LIN {X 29.26, Y 198.76, Z 40.25, A 0, B 90, C 0, E1 0, E2 0, E3 0, E4 0} C_DIS
LIN {X 27.26, Y 190.891, Z 40.25, A 0, B 90, C 0, E1 0, E2 0, E3 0, E4 0} C_DIS
LIN {X 25.335, Y 183.004, Z 40.25, A 0, B 90, C 0, E1 0, E2 0, E3 0, E4 0} C_DIS
LIN {X 23.484, Y 175.099, Z 40.25, A 0, B 90, C 0, E1 0, E2 0, E3 0, E4 0} C_DIS
LIN {X 21.71, Y 167.176, Z 40.25, A 0, B 90, C 0, E1 0, E2 0, E3 0, E4 0} C_DIS
LIN {X 20.012, Y 159.237, Z 40.25, A 0, B 90, C 0, E1 0, E2 0, E3 0, E4 0} C_DIS
LIN {X 18.392, Y 151.282, Z 40.25, A 0, B 90, C 0, E1 0, E2 0, E3 0, E4 0} C_DIS
LIN {X 16.851, Y 143.31, Z 40.25, A 0, B 90, C 0, E1 0, E2 0, E3 0, E4 0} C_DIS
LIN {X 15.39, Y 135.324, Z 40.25, A 0, B 90, C 0, E1 0, E2 0, E3 0, E4 0} C_DIS
LIN {X 14.009, Y 127.324, Z 40.25, A 0, B 90, C 0, E1 0, E2 0, E3 0, E4 0} C_DIS
LIN {X 12.709, Y 119.309, Z 40.25, A 0, B 90, C 0, E1 0, E2 0, E3 0, E4 0} C_DIS
LIN {X 11.491, Y 111.283, Z 40.25, A 0, B 90, C 0, E1 0, E2 0, E3 0, E4 0} C_DIS
LIN {X 10.355, Y 103.244, Z 40.25, A 0, B 90, C 0, E1 0, E2 0, E3 0, E4 0} C_DIS
LIN {X 9.301, Y 95.193, Z 40.25, A 0, B 90, C 0, E1 0, E2 0, E3 0, E4 0} C_DIS
LIN {X 8.331, Y 87.133, Z 40.25, A 0, B 90, C 0, E1 0, E2 0, E3 0, E4 0} C_DIS
LIN {X 7.444, Y 79.063, Z 40.25, A 0, B 90, C 0, E1 0, E2 0, E3 0, E4 0} C_DIS
LIN {X 6.642, Y 70.983, Z 40.25, A 0, B 90, C 0, E1 0, E2 0, E3 0, E4 0} C_DIS
LIN {X 5.924, Y 62.896, Z 40.25, A 0, B 90, C 0, E1 0, E2 0, E3 0, E4 0} C_DIS
LIN {X 5.292, Y 54.802, Z 40.25, A 0, B 90, C 0, E1 0, E2 0, E3 0, E4 0} C_DIS
LIN {X 4.746, Y 46.702, Z 40.25, A 0, B 90, C 0, E1 0, E2 0, E3 0, E4 0} C_DIS
LIN {X 4.285, Y 38.596, Z 40.25, A 0, B 90, C 0, E1 0, E2 0, E3 0, E4 0} C_DIS
LIN {X 3.911, Y 30.486, Z 40.25, A 0, B 90, C 0, E1 0, E2 0, E3 0, E4 0} C_DIS
LIN {X 3.624, Y 22.372, Z 40.25, A 0, B 90, C 0, E1 0, E2 0, E3 0, E4 0} C_DIS
LIN {X 3.424, Y 14.256, Z 40.25, A 0, B 90, C 0, E1 0, E2 0, E3 0, E4 0} C_DIS
LIN {X 3.313, Y 6.138, Z 40.25, A 0, B 90, C 0, E1 0, E2 0, E3 0, E4 0} C_DIS
LIN {X 3.289, Y -1.981, Z 40.25, A 0, B 90, C 0, E1 0, E2 0, E3 0, E4 0} C_DIS
LIN {X 3.353, Y -10.1, Z 40.25, A 0, B 90, C 0, E1 0, E2 0, E3 0, E4 0} C_DIS
LIN {X 3.506, Y -18.217, Z 40.25, A 0, B 90, C 0, E1 0, E2 0, E3 0, E4 0} C_DIS
LIN {X 3.747, Y -26.332, Z 40.25, A 0, B 90, C 0, E1 0, E2 0, E3 0, E4 0} C_DIS
LIN {X 4.074, Y -34.444, Z 40.25, A 0, B 90, C 0, E1 0, E2 0, E3 0, E4 0} C_DIS
LIN {X 4.489, Y -42.553, Z 40.25, A 0, B 90, C 0, E1 0, E2 0, E3 0, E4 0} C_DIS
LIN {X 4.99, Y -50.656, Z 40.25, A 0, B 90, C 0, E1 0, E2 0, E3 0, E4 0} C_DIS
LIN {X 5.578, Y -58.754, Z 40.25, A 0, B 90, C 0, E1 0, E2 0, E3 0, E4 0} C_DIS
LIN {X 6.252, Y -66.844, Z 40.25, A 0, B 90, C 0, E1 0, E2 0, E3 0, E4 0} C_DIS
LIN {X 7.011, Y -74.928, Z 40.25, A 0, B 90, C 0, E1 0, E2 0, E3 0, E4 0} C_DIS
LIN {X 7.855, Y -83.002, Z 40.25, A 0, B 90, C 0, E1 0, E2 0, E3 0, E4 0} C_DIS
LIN {X 8.784, Y -91.068, Z 40.25, A 0, B 90, C 0, E1 0, E2 0, E3 0, E4 0} C_DIS
LIN {X 9.797, Y -99.123, Z 40.25, A 0, B 90, C 0, E1 0, E2 0, E3 0, E4 0} C_DIS
LIN {X 10.893, Y -107.168, Z 40.25, A 0, B 90, C 0, E1 0, E2 0, E3 0, E4 0} C_DIS
LIN {X 12.071, Y -115.201, Z 40.25, A 0, B 90, C 0, E1 0, E2 0, E3 0, E4 0} C_DIS
LIN {X 13.332, Y -123.221, Z 40.25, A 0, B 90, C 0, E1 0, E2 0, E3 0, E4 0} C_DIS
LIN {X 14.674, Y -131.228, Z 40.25, A 0, B 90, C 0, E1 0, E2 0, E3 0, E4 0} C_DIS
LIN {X 16.096, Y -139.221, Z 40.25, A 0, B 90, C 0, E1 0, E2 0, E3 0, E4 0} C_DIS
LIN {X 17.599, Y -147.2, Z 40.25, A 0, B 90, C 0, E1 0, E2 0, E3 0, E4 0} C_DIS
LIN {X 19.18, Y -155.163, Z 40.25, A 0, B 90, C 0, E1 0, E2 0, E3 0, E4 0} C_DIS
LIN {X 20.84, Y -163.111, Z 40.25, A 0, B 90, C 0, E1 0, E2 0, E3 0, E4 0} C_DIS
LIN {X 22.577, Y -171.042, Z 40.25, A 0, B 90, C 0, E1 0, E2 0, E3 0, E4 0} C_DIS
LIN {X 24.389, Y -178.956, Z 40.25, A 0, B 90, C 0, E1 0, E2 0, E3 0, E4 0} C_DIS
LIN {X 26.277, Y -186.852, Z 40.25, A 0, B 90, C 0, E1 0, E2 0, E3 0, E4 0} C_DIS
LIN {X 28.238, Y -194.73, Z 40.25, A 0, B 90, C 0, E1 0, E2 0, E3 0, E4 0} C_DIS
LIN {X 30.272, Y -202.59, Z 40.25, A 0, B 90, C 0, E1 0, E2 0, E3 0, E4 0} C_DIS
LIN {X 32.378, Y -210.431, Z 40.25, A 0, B 90, C 0, E1 0, E2 0, E3 0, E4 0} C_DIS
LIN {X 34.554, Y -218.253, Z 40.25, A 0, B 90, C 0, E1 0, E2 0, E3 0, E4 0} C_DIS
LIN {X 36.8, Y -226.055, Z 40.25, A 0, B 90, C 0, E1 0, E2 0, E3 0, E4 0} C_DIS
LIN {X 39.114, Y -233.837, Z 40.25, A 0, B 90, C 0, E1 0, E2 0, E3 0, E4 0} C_DIS
LIN {X 41.496, Y -241.599, Z 40.25, A 0, B 90, C 0, E1 0, E2 0, E3 0, E4 0} C_DIS
LIN {X 43.943, Y -249.34, Z 40.25, A 0, B 90, C 0, E1 0, E2 0, E3 0, E4 0} C_DIS
LIN {X 46.455, Y -257.06, Z 40.25, A 0, B 90, C 0, E1 0, E2 0, E3 0, E4 0} C_DIS
LIN {X 49.031, Y -264.76, Z 40.25, A 0, B 90, C 0, E1 0, E2 0, E3 0, E4 0} C_DIS
LIN {X 51.67, Y -272.438, Z 40.25, A 0, B 90, C 0, E1 0, E2 0, E3 0, E4 0} C_DIS
LIN {X 54.369, Y -280.094, Z 40.25, A 0, B 90, C 0, E1 0, E2 0, E3 0, E4 0} C_DIS
LIN {X 57.13, Y -287.73, Z 40.25, A 0, B 90, C 0, E1 0, E2 0, E3 0, E4 0} C_DIS
LIN {X 59.951, Y -295.342, Z 40.25, A 0, B 90, C 0, E1 0, E2 0, E3 0, E4 0} C_DIS
LIN {X 62.833, Y -302.932, Z 40.25, A 0, B 90, C 0, E1 0, E2 0, E3 0, E4 0} C_DIS
LIN {X 65.777, Y -310.499, Z 40.25, A 0, B 90, C 0, E1 0, E2 0, E3 0, E4 0} C_DIS
LIN {X 68.781, Y -318.042, Z 40.25, A 0, B 90, C 0, E1 0, E2 0, E3 0, E4 0} C_DIS
LIN {X 71.847, Y -325.559, Z 40.25, A 0, B 90, C 0, E1 0, E2 0, E3 0, E4 0} C_DIS
LIN {X 74.973, Y -333.052, Z 40.25, A 0, B 90, C 0, E1 0, E2 0, E3 0, E4 0} C_DIS
LIN {X 78.074, Y -340.551, Z 40.25, A 0, B 90, C 0, E1 0, E2 0, E3 0, E4 0} C_DIS
LIN {X 75.376, Y -347.755, Z 40.25, A 0, B 90, C 0, E1 0, E2 0, E3 0, E4 0} C_DIS
LIN {X 68.14, Y -351.37, Z 40.25, A 0, B 90, C 0, E1 0, E2 0, E3 0, E4 0} C_DIS
LIN {X 60.675, Y -354.562, Z 40.25, A 0, B 90, C 0, E1 0, E2 0, E3 0, E4 0} C_DIS
LIN {X 53.21, Y -357.754, Z 40.25, A 0, B 90, C 0, E1 0, E2 0, E3 0, E4 0} C_DIS
LIN {X 45.745, Y -360.947, Z 40.25, A 0, B 90, C 0, E1 0, E2 0, E3 0, E4 0} C_DIS
LIN {X 38.28, Y -364.139, Z 40.25, A 0, B 90, C 0, E1 0, E2 0, E3 0, E4 0} C_DIS
LIN {X 30.815, Y -367.331, Z 40.25, A 0, B 90, C 0, E1 0, E2 0, E3 0, E4 0} C_DIS
LIN {X 23.35, Y -370.523, Z 40.25, A 0, B 90, C 0, E1 0, E2 0, E3 0, E4 0} C_DIS
LIN {X 15.615, Y -372.622, Z 40.25, A 0, B 90, C 0, E1 0, E2 0, E3 0, E4 0} C_DIS
LIN {X 9.092, Y -368.331, Z 40.25, A 0, B 90, C 0, E1 0, E2 0, E3 0, E4 0} C_DIS
LIN {X 5.884, Y -360.875, Z 40.25, A 0, B 90, C 0, E1 0, E2 0, E3 0, E4 0} C_DIS
LIN {X 2.773, Y -353.376, Z 40.25, A 0, B 90, C 0, E1 0, E2 0, E3 0, E4 0} C_DIS
LIN {X -0.284, Y -345.854, Z 40.25, A 0, B 90, C 0, E1 0, E2 0, E3 0, E4 0} C_DIS
LIN {X -3.286, Y -338.311, Z 40.25, A 0, B 90, C 0, E1 0, E2 0, E3 0, E4 0} C_DIS
LIN {X -6.234, Y -330.746, Z 40.25, A 0, B 90, C 0, E1 0, E2 0, E3 0, E4 0} C_DIS
LIN {X -9.127, Y -323.16, Z 40.25, A 0, B 90, C 0, E1 0, E2 0, E3 0, E4 0} C_DIS
LIN {X -11.965, Y -315.554, Z 40.25, A 0, B 90, C 0, E1 0, E2 0, E3 0, E4 0} C_DIS
LIN {X -14.749, Y -307.927, Z 40.25, A 0, B 90, C 0, E1 0, E2 0, E3 0, E4 0} C_DIS
LIN {X -17.478, Y -300.281, Z 40.25, A 0, B 90, C 0, E1 0, E2 0, E3 0, E4 0} C_DIS
LIN {X -20.15, Y -292.614, Z 40.25, A 0, B 90, C 0, E1 0, E2 0, E3 0, E4 0} C_DIS
LIN {X -22.764, Y -284.928, Z 40.25, A 0, B 90, C 0, E1 0, E2 0, E3 0, E4 0} C_DIS
LIN {X -25.32, Y -277.221, Z 40.25, A 0, B 90, C 0, E1 0, E2 0, E3 0, E4 0} C_DIS
LIN {X -27.815, Y -269.496, Z 40.25, A 0, B 90, C 0, E1 0, E2 0, E3 0, E4 0} C_DIS
LIN {X -30.249, Y -261.75, Z 40.25, A 0, B 90, C 0, E1 0, E2 0, E3 0, E4 0} C_DIS
LIN {X -32.621, Y -253.986, Z 40.25, A 0, B 90, C 0, E1 0, E2 0, E3 0, E4 0} C_DIS
LIN {X -34.93, Y -246.202, Z 40.25, A 0, B 90, C 0, E1 0, E2 0, E3 0, E4 0} C_DIS
LIN {X -37.174, Y -238.399, Z 40.25, A 0, B 90, C 0, E1 0, E2 0, E3 0, E4 0} C_DIS
LIN {X -39.353, Y -230.578, Z 40.25, A 0, B 90, C 0, E1 0, E2 0, E3 0, E4 0} C_DIS
LIN {X -41.465, Y -222.739, Z 40.25, A 0, B 90, C 0, E1 0, E2 0, E3 0, E4 0} C_DIS
LIN {X -43.512, Y -214.883, Z 40.25, A 0, B 90, C 0, E1 0, E2 0, E3 0, E4 0} C_DIS
LIN {X -45.49, Y -207.009, Z 40.25, A 0, B 90, C 0, E1 0, E2 0, E3 0, E4 0} C_DIS
LIN {X -47.401, Y -199.118, Z 40.25, A 0, B 90, C 0, E1 0, E2 0, E3 0, E4 0} C_DIS
LIN {X -49.243, Y -191.211, Z 40.25, A 0, B 90, C 0, E1 0, E2 0, E3 0, E4 0} C_DIS
LIN {X -51.015, Y -183.288, Z 40.25, A 0, B 90, C 0, E1 0, E2 0, E3 0, E4 0} C_DIS
LIN {X -52.717, Y -175.349, Z 40.25, A 0, B 90, C 0, E1 0, E2 0, E3 0, E4 0} C_DIS
LIN {X -54.348, Y -167.396, Z 40.25, A 0, B 90, C 0, E1 0, E2 0, E3 0, E4 0} C_DIS
LIN {X -55.907, Y -159.428, Z 40.25, A 0, B 90, C 0, E1 0, E2 0, E3 0, E4 0} C_DIS
LIN {X -57.394, Y -151.446, Z 40.25, A 0, B 90, C 0, E1 0, E2 0, E3 0, E4 0} C_DIS
LIN {X -58.807, Y -143.452, Z 40.25, A 0, B 90, C 0, E1 0, E2 0, E3 0, E4 0} C_DIS
LIN {X -60.147, Y -135.444, Z 40.25, A 0, B 90, C 0, E1 0, E2 0, E3 0, E4 0} C_DIS
LIN {X -61.412, Y -127.424, Z 40.25, A 0, B 90, C 0, E1 0, E2 0, E3 0, E4 0} C_DIS
LIN {X -62.602, Y -119.393, Z 40.25, A 0, B 90, C 0, E1 0, E2 0, E3 0, E4 0} C_DIS
LIN {X -63.717, Y -111.351, Z 40.25, A 0, B 90, C 0, E1 0, E2 0, E3 0, E4 0} C_DIS
LIN {X -64.755, Y -103.299, Z 40.25, A 0, B 90, C 0, E1 0, E2 0, E3 0, E4 0} C_DIS
LIN {X -65.718, Y -95.238, Z 40.25, A 0, B 90, C 0, E1 0, E2 0, E3 0, E4 0} C_DIS
LIN {X -66.604, Y -87.167, Z 40.25, A 0, B 90, C 0, E1 0, E2 0, E3 0, E4 0} C_DIS
LIN {X -67.412, Y -79.089, Z 40.25, A 0, B 90, C 0, E1 0, E2 0, E3 0, E4 0} C_DIS
LIN {X -68.144, Y -71.003, Z 40.25, A 0, B 90, C 0, E1 0, E2 0, E3 0, E4 0} C_DIS
LIN {X -68.798, Y -62.911, Z 40.25, A 0, B 90, C 0, E1 0, E2 0, E3 0, E4 0} C_DIS
LIN {X -69.374, Y -54.812, Z 40.25, A 0, B 90, C 0, E1 0, E2 0, E3 0, E4 0} C_DIS
LIN {X -69.872, Y -46.709, Z 40.25, A 0, B 90, C 0, E1 0, E2 0, E3 0, E4 0} C_DIS
LIN {X -70.291, Y -38.601, Z 40.25, A 0, B 90, C 0, E1 0, E2 0, E3 0, E4 0} C_DIS
LIN {X -70.631, Y -30.489, Z 40.25, A 0, B 90, C 0, E1 0, E2 0, E3 0, E4 0} C_DIS
LIN {X -70.892, Y -22.374, Z 40.25, A 0, B 90, C 0, E1 0, E2 0, E3 0, E4 0} C_DIS
LIN {X -71.073, Y -14.257, Z 40.25, A 0, B 90, C 0, E1 0, E2 0, E3 0, E4 0} C_DIS
LIN {X -71.174, Y -6.139, Z 40.25, A 0, B 90, C 0, E1 0, E2 0, E3 0, E4 0} C_DIS
LIN {X -71.195, Y 1.979, Z 40.25, A 0, B 90, C 0, E1 0, E2 0, E3 0, E4 0} C_DIS
LIN {X -71.136, Y 10.098, Z 40.25, A 0, B 90, C 0, E1 0, E2 0, E3 0, E4 0} C_DIS
LIN {X -70.996, Y 18.216, Z 40.25, A 0, B 90, C 0, E1 0, E2 0, E3 0, E4 0} C_DIS
LIN {X -70.777, Y 26.332, Z 40.25, A 0, B 90, C 0, E1 0, E2 0, E3 0, E4 0} C_DIS
LIN {X -70.478, Y 34.445, Z 40.25, A 0, B 90, C 0, E1 0, E2 0, E3 0, E4 0} C_DIS
LIN {X -70.099, Y 42.555, Z 40.25, A 0, B 90, C 0, E1 0, E2 0, E3 0, E4 0} C_DIS
LIN {X -69.642, Y 50.661, Z 40.25, A 0, B 90, C 0, E1 0, E2 0, E3 0, E4 0} C_DIS
LIN {X -69.107, Y 58.762, Z 40.25, A 0, B 90, C 0, E1 0, E2 0, E3 0, E4 0} C_DIS
LIN {X -68.493, Y 66.858, Z 40.25, A 0, B 90, C 0, E1 0, E2 0, E3 0, E4 0} C_DIS
LIN {X -67.801, Y 74.947, Z 40.25, A 0, B 90, C 0, E1 0, E2 0, E3 0, E4 0} C_DIS
LIN {X -67.031, Y 83.029, Z 40.25, A 0, B 90, C 0, E1 0, E2 0, E3 0, E4 0} C_DIS
LIN {X -66.184, Y 91.104, Z 40.25, A 0, B 90, C 0, E1 0, E2 0, E3 0, E4 0} C_DIS
LIN {X -65.26, Y 99.17, Z 40.25, A 0, B 90, C 0, E1 0, E2 0, E3 0, E4 0} C_DIS
LIN {X -64.26, Y 107.227, Z 40.25, A 0, B 90, C 0, E1 0, E2 0, E3 0, E4 0} C_DIS
LIN {X -63.183, Y 115.274, Z 40.25, A 0, B 90, C 0, E1 0, E2 0, E3 0, E4 0} C_DIS
LIN {X -62.031, Y 123.311, Z 40.25, A 0, B 90, C 0, E1 0, E2 0, E3 0, E4 0} C_DIS
LIN {X -60.803, Y 131.336, Z 40.25, A 0, B 90, C 0, E1 0, E2 0, E3 0, E4 0} C_DIS
LIN {X -59.501, Y 139.35, Z 40.25, A 0, B 90, C 0, E1 0, E2 0, E3 0, E4 0} C_DIS
LIN {X -58.125, Y 147.351, Z 40.25, A 0, B 90, C 0, E1 0, E2 0, E3 0, E4 0} C_DIS
LIN {X -56.675, Y 155.339, Z 40.25, A 0, B 90, C 0, E1 0, E2 0, E3 0, E4 0} C_DIS
LIN {X -55.153, Y 163.314, Z 40.25, A 0, B 90, C 0, E1 0, E2 0, E3 0, E4 0} C_DIS
LIN {X -53.558, Y 171.275, Z 40.25, A 0, B 90, C 0, E1 0, E2 0, E3 0, E4 0} C_DIS
LIN {X -51.893, Y 179.221, Z 40.25, A 0, B 90, C 0, E1 0, E2 0, E3 0, E4 0} C_DIS
LIN {X -50.157, Y 187.152, Z 40.25, A 0, B 90, C 0, E1 0, E2 0, E3 0, E4 0} C_DIS
LIN {X -48.351, Y 195.068, Z 40.25, A 0, B 90, C 0, E1 0, E2 0, E3 0, E4 0} C_DIS
LIN {X -46.476, Y 202.967, Z 40.25, A 0, B 90, C 0, E1 0, E2 0, E3 0, E4 0} C_DIS
LIN {X -44.533, Y 210.85, Z 40.25, A 0, B 90, C 0, E1 0, E2 0, E3 0, E4 0} C_DIS
LIN {X -42.521, Y 218.716, Z 40.25, A 0, B 90, C 0, E1 0, E2 0, E3 0, E4 0} C_DIS
LIN {X -40.443, Y 226.564, Z 40.25, A 0, B 90, C 0, E1 0, E2 0, E3 0, E4 0} C_DIS
LIN {X -38.298, Y 234.394, Z 40.25, A 0, B 90, C 0, E1 0, E2 0, E3 0, E4 0} C_DIS
LIN {X -36.088, Y 242.206, Z 40.25, A 0, B 90, C 0, E1 0, E2 0, E3 0, E4 0} C_DIS
LIN {X -34.098, Y 250, Z 42.75, A 0, B 90, C 0, E1 0, E2 0, E3 0, E4 0} C_DIS
LIN {X -31.758, Y 257.753, Z 42.75, A 0, B 90, C 0, E1 0, E2 0, E3 0, E4 0} C_DIS
LIN {X -29.355, Y 265.488, Z 42.75, A 0, B 90, C 0, E1 0, E2 0, E3 0, E4 0} C_DIS
LIN {X -26.891, Y 273.202, Z 42.75, A 0, B 90, C 0, E1 0, E2 0, E3 0, E4 0} C_DIS
LIN {X -24.365, Y 280.897, Z 42.75, A 0, B 90, C 0, E1 0, E2 0, E3 0, E4 0} C_DIS
LIN {X -21.781, Y 288.573, Z 42.75, A 0, B 90, C 0, E1 0, E2 0, E3 0, E4 0} C_DIS
LIN {X -19.138, Y 296.228, Z 42.75, A 0, B 90, C 0, E1 0, E2 0, E3 0, E4 0} C_DIS
LIN {X -16.439, Y 303.864, Z 42.75, A 0, B 90, C 0, E1 0, E2 0, E3 0, E4 0} C_DIS
LIN {X -13.684, Y 311.48, Z 42.75, A 0, B 90, C 0, E1 0, E2 0, E3 0, E4 0} C_DIS
LIN {X -10.874, Y 319.076, Z 42.75, A 0, B 90, C 0, E1 0, E2 0, E3 0, E4 0} C_DIS
LIN {X -8.01, Y 326.652, Z 42.75, A 0, B 90, C 0, E1 0, E2 0, E3 0, E4 0} C_DIS
LIN {X -5.092, Y 334.206, Z 42.75, A 0, B 90, C 0, E1 0, E2 0, E3 0, E4 0} C_DIS
LIN {X -2.12, Y 341.74, Z 42.75, A 0, B 90, C 0, E1 0, E2 0, E3 0, E4 0} C_DIS
LIN {X 0.906, Y 349.252, Z 42.75, A 0, B 90, C 0, E1 0, E2 0, E3 0, E4 0} C_DIS
LIN {X 3.988, Y 356.742, Z 42.75, A 0, B 90, C 0, E1 0, E2 0, E3 0, E4 0} C_DIS
LIN {X 7.123, Y 364.209, Z 42.75, A 0, B 90, C 0, E1 0, E2 0, E3 0, E4 0} C_DIS
LIN {X 11.532, Y 370.814, Z 42.75, A 0, B 90, C 0, E1 0, E2 0, E3 0, E4 0} C_DIS
LIN {X 19.315, Y 371.572, Z 42.75, A 0, B 90, C 0, E1 0, E2 0, E3 0, E4 0} C_DIS
LIN {X 26.761, Y 368.386, Z 42.75, A 0, B 90, C 0, E1 0, E2 0, E3 0, E4 0} C_DIS
LIN {X 34.207, Y 365.2, Z 42.75, A 0, B 90, C 0, E1 0, E2 0, E3 0, E4 0} C_DIS
LIN {X 41.653, Y 362.015, Z 42.75, A 0, B 90, C 0, E1 0, E2 0, E3 0, E4 0} C_DIS
LIN {X 49.099, Y 358.829, Z 42.75, A 0, B 90, C 0, E1 0, E2 0, E3 0, E4 0} C_DIS
LIN {X 56.545, Y 355.643, Z 42.75, A 0, B 90, C 0, E1 0, E2 0, E3 0, E4 0} C_DIS
LIN {X 63.991, Y 352.457, Z 42.75, A 0, B 90, C 0, E1 0, E2 0, E3 0, E4 0} C_DIS
LIN {X 71.413, Y 349.22, Z 42.75, A 0, B 90, C 0, E1 0, E2 0, E3 0, E4 0} C_DIS
LIN {X 76.279, Y 343.133, Z 42.75, A 0, B 90, C 0, E1 0, E2 0, E3 0, E4 0} C_DIS
LIN {X 74.034, Y 335.474, Z 42.75, A 0, B 90, C 0, E1 0, E2 0, E3 0, E4 0} C_DIS
LIN {X 70.897, Y 328.008, Z 42.75, A 0, B 90, C 0, E1 0, E2 0, E3 0, E4 0} C_DIS
LIN {X 67.819, Y 320.517, Z 42.75, A 0, B 90, C 0, E1 0, E2 0, E3 0, E4 0} C_DIS
LIN {X 64.802, Y 313.001, Z 42.75, A 0, B 90, C 0, E1 0, E2 0, E3 0, E4 0} C_DIS
LIN {X 61.845, Y 305.461, Z 42.75, A 0, B 90, C 0, E1 0, E2 0, E3 0, E4 0} C_DIS
LIN {X 58.948, Y 297.898, Z 42.75, A 0, B 90, C 0, E1 0, E2 0, E3 0, E4 0} C_DIS
LIN {X 56.111, Y 290.312, Z 42.75, A 0, B 90, C 0, E1 0, E2 0, E3 0, E4 0} C_DIS
LIN {X 53.332, Y 282.705, Z 42.75, A 0, B 90, C 0, E1 0, E2 0, E3 0, E4 0} C_DIS
LIN {X 50.614, Y 275.076, Z 42.75, A 0, B 90, C 0, E1 0, E2 0, E3 0, E4 0} C_DIS
LIN {X 47.955, Y 267.426, Z 42.75, A 0, B 90, C 0, E1 0, E2 0, E3 0, E4 0} C_DIS
LIN {X 45.357, Y 259.755, Z 42.75, A 0, B 90, C 0, E1 0, E2 0, E3 0, E4 0} C_DIS
LIN {X 42.821, Y 252.064, Z 42.75, A 0, B 90, C 0, E1 0, E2 0, E3 0, E4 0} C_DIS
LIN {X 40.35, Y 244.351, Z 42.75, A 0, B 90, C 0, E1 0, E2 0, E3 0, E4 0} C_DIS
LIN {X 37.943, Y 236.618, Z 42.75, A 0, B 90, C 0, E1 0, E2 0, E3 0, E4 0} C_DIS
LIN {X 35.604, Y 228.864, Z 42.75, A 0, B 90, C 0, E1 0, E2 0, E3 0, E4 0} C_DIS
LIN {X 33.332, Y 221.091, Z 42.75, A 0, B 90, C 0, E1 0, E2 0, E3 0, E4 0} C_DIS
LIN {X 31.13, Y 213.297, Z 42.75, A 0, B 90, C 0, E1 0, E2 0, E3 0, E4 0} C_DIS
LIN {X 28.998, Y 205.484, Z 42.75, A 0, B 90, C 0, E1 0, E2 0, E3 0, E4 0} C_DIS
LIN {X 26.939, Y 197.651, Z 42.75, A 0, B 90, C 0, E1 0, E2 0, E3 0, E4 0} C_DIS
LIN {X 24.952, Y 189.8, Z 42.75, A 0, B 90, C 0, E1 0, E2 0, E3 0, E4 0} C_DIS
LIN {X 23.04, Y 181.93, Z 42.75, A 0, B 90, C 0, E1 0, E2 0, E3 0, E4 0} C_DIS
LIN {X 21.202, Y 174.042, Z 42.75, A 0, B 90, C 0, E1 0, E2 0, E3 0, E4 0} C_DIS
LIN {X 19.439, Y 166.137, Z 42.75, A 0, B 90, C 0, E1 0, E2 0, E3 0, E4 0} C_DIS
LIN {X 17.754, Y 158.216, Z 42.75, A 0, B 90, C 0, E1 0, E2 0, E3 0, E4 0} C_DIS
LIN {X 16.146, Y 150.278, Z 42.75, A 0, B 90, C 0, E1 0, E2 0, E3 0, E4 0} C_DIS
LIN {X 14.617, Y 142.325, Z 42.75, A 0, B 90, C 0, E1 0, E2 0, E3 0, E4 0} C_DIS
LIN {X 13.168, Y 134.357, Z 42.75, A 0, B 90, C 0, E1 0, E2 0, E3 0, E4 0} C_DIS
LIN {X 11.799, Y 126.375, Z 42.75, A 0, B 90, C 0, E1 0, E2 0, E3 0, E4 0} C_DIS
LIN {X 10.51, Y 118.379, Z 42.75, A 0, B 90, C 0, E1 0, E2 0, E3 0, E4 0} C_DIS
LIN {X 9.303, Y 110.371, Z 42.75, A 0, B 90, C 0, E1 0, E2 0, E3 0, E4 0} C_DIS
LIN {X 8.178, Y 102.35, Z 42.75, A 0, B 90, C 0, E1 0, E2 0, E3 0, E4 0} C_DIS
LIN {X 7.135, Y 94.319, Z 42.75, A 0, B 90, C 0, E1 0, E2 0, E3 0, E4 0} C_DIS
LIN {X 6.175, Y 86.277, Z 42.75, A 0, B 90, C 0, E1 0, E2 0, E3 0, E4 0} C_DIS
LIN {X 5.298, Y 78.226, Z 42.75, A 0, B 90, C 0, E1 0, E2 0, E3 0, E4 0} C_DIS
LIN {X 4.506, Y 70.166, Z 42.75, A 0, B 90, C 0, E1 0, E2 0, E3 0, E4 0} C_DIS
LIN {X 3.798, Y 62.098, Z 42.75, A 0, B 90, C 0, E1 0, E2 0, E3 0, E4 0} C_DIS
LIN {X 3.175, Y 54.023, Z 42.75, A 0, B 90, C 0, E1 0, E2 0, E3 0, E4 0} C_DIS
LIN {X 2.637, Y 45.942, Z 42.75, A 0, B 90, C 0, E1 0, E2 0, E3 0, E4 0} C_DIS
LIN {X 2.185, Y 37.856, Z 42.75, A 0, B 90, C 0, E1 0, E2 0, E3 0, E4 0} C_DIS
LIN {X 1.82, Y 29.766, Z 42.75, A 0, B 90, C 0, E1 0, E2 0, E3 0, E4 0} C_DIS
LIN {X 1.541, Y 21.672, Z 42.75, A 0, B 90, C 0, E1 0, E2 0, E3 0, E4 0} C_DIS
LIN {X 1.349, Y 13.575, Z 42.75, A 0, B 90, C 0, E1 0, E2 0, E3 0, E4 0} C_DIS
LIN {X 1.244, Y 5.477, Z 42.75, A 0, B 90, C 0, E1 0, E2 0, E3 0, E4 0} C_DIS
LIN {X 1.227, Y -2.622, Z 42.75, A 0, B 90, C 0, E1 0, E2 0, E3 0, E4 0} C_DIS
LIN {X 1.299, Y -10.721, Z 42.75, A 0, B 90, C 0, E1 0, E2 0, E3 0, E4 0} C_DIS
LIN {X 1.458, Y -18.818, Z 42.75, A 0, B 90, C 0, E1 0, E2 0, E3 0, E4 0} C_DIS
LIN {X 1.704, Y -26.913, Z 42.75, A 0, B 90, C 0, E1 0, E2 0, E3 0, E4 0} C_DIS
LIN {X 2.037, Y -35.005, Z 42.75, A 0, B 90, C 0, E1 0, E2 0, E3 0, E4 0} C_DIS
LIN {X 2.457, Y -43.093, Z 42.75, A 0, B 90, C 0, E1 0, E2 0, E3 0, E4 0} C_DIS
LIN {X 2.963, Y -51.176, Z 42.75, A 0, B 90, C 0, E1 0, E2 0, E3 0, E4 0} C_DIS
LIN {X 3.555, Y -59.253, Z 42.75, A 0, B 90, C 0, E1 0, E2 0, E3 0, E4 0} C_DIS
LIN {X 4.233, Y -67.323, Z 42.75, A 0, B 90, C 0, E1 0, E2 0, E3 0, E4 0} C_DIS
LIN {X 4.996, Y -75.386, Z 42.75, A 0, B 90, C 0, E1 0, E2 0, E3 0, E4 0} C_DIS
LIN {X 5.844, Y -83.441, Z 42.75, A 0, B 90, C 0, E1 0, E2 0, E3 0, E4 0} C_DIS
LIN {X 6.776, Y -91.486, Z 42.75, A 0, B 90, C 0, E1 0, E2 0, E3 0, E4 0} C_DIS
LIN {X 7.792, Y -99.52, Z 42.75, A 0, B 90, C 0, E1 0, E2 0, E3 0, E4 0} C_DIS
LIN {X 8.89, Y -107.544, Z 42.75, A 0, B 90, C 0, E1 0, E2 0, E3 0, E4 0} C_DIS
LIN {X 10.071, Y -115.557, Z 42.75, A 0, B 90, C 0, E1 0, E2 0, E3 0, E4 0} C_DIS
LIN {X 11.334, Y -123.557, Z 42.75, A 0, B 90, C 0, E1 0, E2 0, E3 0, E4 0} C_DIS
LIN {X 12.677, Y -131.543, Z 42.75, A 0, B 90, C 0, E1 0, E2 0, E3 0, E4 0} C_DIS
LIN {X 14.101, Y -139.516, Z 42.75, A 0, B 90, C 0, E1 0, E2 0, E3 0, E4 0} C_DIS
LIN {X 15.604, Y -147.474, Z 42.75, A 0, B 90, C 0, E1 0, E2 0, E3 0, E4 0} C_DIS
LIN {X 17.186, Y -155.417, Z 42.75, A 0, B 90, C 0, E1 0, E2 0, E3 0, E4 0} C_DIS
LIN {X 18.846, Y -163.344, Z 42.75, A 0, B 90, C 0, E1 0, E2 0, E3 0, E4 0} C_DIS
LIN {X 20.583, Y -171.254, Z 42.75, A 0, B 90, C 0, E1 0, E2 0, E3 0, E4 0} C_DIS
LIN {X 22.395, Y -179.148, Z 42.75, A 0, B 90, C 0, E1 0, E2 0, E3 0, E4 0} C_DIS
LIN {X 24.282, Y -187.024, Z 42.75, A 0, B 90, C 0, E1 0, E2 0, E3 0, E4 0} C_DIS
LIN {X 26.242, Y -194.882, Z 42.75, A 0, B 90, C 0, E1 0, E2 0, E3 0, E4 0} C_DIS
LIN {X 28.275, Y -202.721, Z 42.75, A 0, B 90, C 0, E1 0, E2 0, E3 0, E4 0} C_DIS
LIN {X 30.379, Y -210.542, Z 42.75, A 0, B 90, C 0, E1 0, E2 0, E3 0, E4 0} C_DIS
LIN {X 32.553, Y -218.344, Z 42.75, A 0, B 90, C 0, E1 0, E2 0, E3 0, E4 0} C_DIS
LIN {X 34.796, Y -226.126, Z 42.75, A 0, B 90, C 0, E1 0, E2 0, E3 0, E4 0} C_DIS
LIN {X 37.107, Y -233.888, Z 42.75, A 0, B 90, C 0, E1 0, E2 0, E3 0, E4 0} C_DIS
LIN {X 39.485, Y -241.63, Z 42.75, A 0, B 90, C 0, E1 0, E2 0, E3 0, E4 0} C_DIS
LIN {X 41.929, Y -249.351, Z 42.75, A 0, B 90, C 0, E1 0, E2 0, E3 0, E4 0} C_DIS
LIN {X 44.438, Y -257.052, Z 42.75, A 0, B 90, C 0, E1 0, E2 0, E3 0, E4 0} C_DIS
LIN {X 47.009, Y -264.731, Z 42.75, A 0, B 90, C 0, E1 0, E2 0, E3 0, E4 0} C_DIS
LIN {X 49.644, Y -272.39, Z 42.75, A 0, B 90, C 0, E1 0, E2 0, E3 0, E4 0} C_DIS
LIN {X 52.339, Y -280.027, Z 42.75, A 0, B 90, C 0, E1 0, E2 0, E3 0, E4 0} C_DIS
LIN {X 55.096, Y -287.642, Z 42.75, A 0, B 90, C 0, E1 0, E2 0, E3 0, E4 0} C_DIS
LIN {X 57.912, Y -295.235, Z 42.75, A 0, B 90, C 0, E1 0, E2 0, E3 0, E4 0} C_DIS
LIN {X 60.79, Y -302.806, Z 42.75, A 0, B 90, C 0, E1 0, E2 0, E3 0, E4 0} C_DIS
LIN {X 63.728, Y -310.353, Z 42.75, A 0, B 90, C 0, E1 0, E2 0, E3 0, E4 0} C_DIS
LIN {X 66.727, Y -317.876, Z 42.75, A 0, B 90, C 0, E1 0, E2 0, E3 0, E4 0} C_DIS
LIN {X 69.788, Y -325.374, Z 42.75, A 0, B 90, C 0, E1 0, E2 0, E3 0, E4 0} C_DIS
LIN {X 72.909, Y -332.848, Z 42.75, A 0, B 90, C 0, E1 0, E2 0, E3 0, E4 0} C_DIS
LIN {X 76.053, Y -340.31, Z 42.75, A 0, B 90, C 0, E1 0, E2 0, E3 0, E4 0} C_DIS
LIN {X 73.764, Y -347.619, Z 42.75, A 0, B 90, C 0, E1 0, E2 0, E3 0, E4 0} C_DIS
LIN {X 66.616, Y -351.338, Z 42.75, A 0, B 90, C 0, E1 0, E2 0, E3 0, E4 0} C_DIS
LIN {X 59.17, Y -354.523, Z 42.75, A 0, B 90, C 0, E1 0, E2 0, E3 0, E4 0} C_DIS
LIN {X 51.724, Y -357.709, Z 42.75, A 0, B 90, C 0, E1 0, E2 0, E3 0, E4 0} C_DIS
LIN {X 44.278, Y -360.895, Z 42.75, A 0, B 90, C 0, E1 0, E2 0, E3 0, E4 0} C_DIS
LIN {X 36.832, Y -364.081, Z 42.75, A 0, B 90, C 0, E1 0, E2 0, E3 0, E4 0} C_DIS
LIN {X 29.386, Y -367.266, Z 42.75, A 0, B 90, C 0, E1 0, E2 0, E3 0, E4 0} C_DIS
LIN {X 21.94, Y -370.452, Z 42.75, A 0, B 90, C 0, E1 0, E2 0, E3 0, E4 0} C_DIS
LIN {X 14.148, Y -371.925, Z 42.75, A 0, B 90, C 0, E1 0, E2 0, E3 0, E4 0} C_DIS
LIN {X 8.242, Y -366.839, Z 42.75, A 0, B 90, C 0, E1 0, E2 0, E3 0, E4 0} C_DIS
LIN {X 5.087, Y -359.38, Z 42.75, A 0, B 90, C 0, E1 0, E2 0, E3 0, E4 0} C_DIS
LIN {X 1.986, Y -351.898, Z 42.75, A 0, B 90, C 0, E1 0, E2 0, E3 0, E4 0} C_DIS
LIN {X -1.06, Y -344.394, Z 42.75, A 0, B 90, C 0, E1 0, E2 0, E3 0, E4 0} C_DIS
LIN {X -4.052, Y -336.868, Z 42.75, A 0, B 90, C 0, E1 0, E2 0, E3 0, E4 0} C_DIS
LIN {X -6.989, Y -329.32, Z 42.75, A 0, B 90, C 0, E1 0, E2 0, E3 0, E4 0} C_DIS
LIN {X -9.872, Y -321.752, Z 42.75, A 0, B 90, C 0, E1 0, E2 0, E3 0, E4 0} C_DIS
LIN {X -12.7, Y -314.163, Z 42.75, A 0, B 90, C 0, E1 0, E2 0, E3 0, E4 0} C_DIS
LIN {X -15.474, Y -306.554, Z 42.75, A 0, B 90, C 0, E1 0, E2 0, E3 0, E4 0} C_DIS
LIN {X -18.193, Y -298.925, Z 42.75, A 0, B 90, C 0, E1 0, E2 0, E3 0, E4 0} C_DIS
LIN {X -20.855, Y -291.277, Z 42.75, A 0, B 90, C 0, E1 0, E2 0, E3 0, E4 0} C_DIS
LIN {X -23.46, Y -283.608, Z 42.75, A 0, B 90, C 0, E1 0, E2 0, E3 0, E4 0} C_DIS
LIN {X -26.006, Y -275.92, Z 42.75, A 0, B 90, C 0, E1 0, E2 0, E3 0, E4 0} C_DIS
LIN {X -28.492, Y -268.212, Z 42.75, A 0, B 90, C 0, E1 0, E2 0, E3 0, E4 0} C_DIS
LIN {X -30.917, Y -260.485, Z 42.75, A 0, B 90, C 0, E1 0, E2 0, E3 0, E4 0} C_DIS
LIN {X -33.279, Y -252.738, Z 42.75, A 0, B 90, C 0, E1 0, E2 0, E3 0, E4 0} C_DIS
LIN {X -35.578, Y -244.972, Z 42.75, A 0, B 90, C 0, E1 0, E2 0, E3 0, E4 0} C_DIS
LIN {X -37.812, Y -237.188, Z 42.75, A 0, B 90, C 0, E1 0, E2 0, E3 0, E4 0} C_DIS
LIN {X -39.982, Y -229.385, Z 42.75, A 0, B 90, C 0, E1 0, E2 0, E3 0, E4 0} C_DIS
LIN {X -42.085, Y -221.564, Z 42.75, A 0, B 90, C 0, E1 0, E2 0, E3 0, E4 0} C_DIS
LIN {X -44.122, Y -213.725, Z 42.75, A 0, B 90, C 0, E1 0, E2 0, E3 0, E4 0} C_DIS
LIN {X -46.092, Y -205.87, Z 42.75, A 0, B 90, C 0, E1 0, E2 0, E3 0, E4 0} C_DIS
LIN {X -47.994, Y -197.997, Z 42.75, A 0, B 90, C 0, E1 0, E2 0, E3 0, E4 0} C_DIS
LIN {X -49.826, Y -190.108, Z 42.75, A 0, B 90, C 0, E1 0, E2 0, E3 0, E4 0} C_DIS
LIN {X -51.589, Y -182.204, Z 42.75, A 0, B 90, C 0, E1 0, E2 0, E3 0, E4 0} C_DIS
LIN {X -53.282, Y -174.284, Z 42.75, A 0, B 90, C 0, E1 0, E2 0, E3 0, E4 0} C_DIS
LIN {X -54.904, Y -166.349, Z 42.75, A 0, B 90, C 0, E1 0, E2 0, E3 0, E4 0} C_DIS
LIN {X -56.455, Y -158.4, Z 42.75, A 0, B 90, C 0, E1 0, E2 0, E3 0, E4 0} C_DIS
LIN {X -57.932, Y -150.437, Z 42.75, A 0, B 90, C 0, E1 0, E2 0, E3 0, E4 0} C_DIS
LIN {X -59.337, Y -142.461, Z 42.75, A 0, B 90, C 0, E1 0, E2 0, E3 0, E4 0} C_DIS
LIN {X -60.668, Y -134.472, Z 42.75, A 0, B 90, C 0, E1 0, E2 0, E3 0, E4 0} C_DIS
LIN {X -61.925, Y -126.472, Z 42.75, A 0, B 90, C 0, E1 0, E2 0, E3 0, E4 0} C_DIS
LIN {X -63.107, Y -118.459, Z 42.75, A 0, B 90, C 0, E1 0, E2 0, E3 0, E4 0} C_DIS
LIN {X -64.213, Y -110.437, Z 42.75, A 0, B 90, C 0, E1 0, E2 0, E3 0, E4 0} C_DIS
LIN {X -65.244, Y -102.404, Z 42.75, A 0, B 90, C 0, E1 0, E2 0, E3 0, E4 0} C_DIS
LIN {X -66.198, Y -94.361, Z 42.75, A 0, B 90, C 0, E1 0, E2 0, E3 0, E4 0} C_DIS
LIN {X -67.076, Y -86.31, Z 42.75, A 0, B 90, C 0, E1 0, E2 0, E3 0, E4 0} C_DIS
LIN {X -67.878, Y -78.251, Z 42.75, A 0, B 90, C 0, E1 0, E2 0, E3 0, E4 0} C_DIS
LIN {X -68.602, Y -70.185, Z 42.75, A 0, B 90, C 0, E1 0, E2 0, E3 0, E4 0} C_DIS
LIN {X -69.248, Y -62.112, Z 42.75, A 0, B 90, C 0, E1 0, E2 0, E3 0, E4 0} C_DIS
LIN {X -69.817, Y -54.033, Z 42.75, A 0, B 90, C 0, E1 0, E2 0, E3 0, E4 0} C_DIS
LIN {X -70.308, Y -45.949, Z 42.75, A 0, B 90, C 0, E1 0, E2 0, E3 0, E4 0} C_DIS
LIN {X -70.72, Y -37.86, Z 42.75, A 0, B 90, C 0, E1 0, E2 0, E3 0, E4 0} C_DIS
LIN {X -71.053, Y -29.768, Z 42.75, A 0, B 90, C 0, E1 0, E2 0, E3 0, E4 0} C_DIS
LIN {X -71.307, Y -21.674, Z 42.75, A 0, B 90, C 0, E1 0, E2 0, E3 0, E4 0} C_DIS
LIN {X -71.482, Y -13.577, Z 42.75, A 0, B 90, C 0, E1 0, E2 0, E3 0, E4 0} C_DIS
LIN {X -71.577, Y -5.478, Z 42.75, A 0, B 90, C 0, E1 0, E2 0, E3 0, E4 0} C_DIS
LIN {X -71.591, Y 2.621, Z 42.75, A 0, B 90, C 0, E1 0, E2 0, E3 0, E4 0} C_DIS
LIN {X -71.525, Y 10.719, Z 42.75, A 0, B 90, C 0, E1 0, E2 0, E3 0, E4 0} C_DIS
LIN {X -71.38, Y 18.817, Z 42.75, A 0, B 90, C 0, E1 0, E2 0, E3 0, E4 0} C_DIS
LIN {X -71.154, Y 26.912, Z 42.75, A 0, B 90, C 0, E1 0, E2 0, E3 0, E4 0} C_DIS
LIN {X -70.849, Y 35.005, Z 42.75, A 0, B 90, C 0, E1 0, E2 0, E3 0, E4 0} C_DIS
LIN {X -70.465, Y 43.095, Z 42.75, A 0, B 90, C 0, E1 0, E2 0, E3 0, E4 0} C_DIS
LIN {X -70.003, Y 51.181, Z 42.75, A 0, B 90, C 0, E1 0, E2 0, E3 0, E4 0} C_DIS
LIN {X -69.462, Y 59.262, Z 42.75, A 0, B 90, C 0, E1 0, E2 0, E3 0, E4 0} C_DIS
LIN {X -68.843, Y 67.337, Z 42.75, A 0, B 90, C 0, E1 0, E2 0, E3 0, E4 0} C_DIS
LIN {X -68.146, Y 75.406, Z 42.75, A 0, B 90, C 0, E1 0, E2 0, E3 0, E4 0} C_DIS
LIN {X -67.372, Y 83.467, Z 42.75, A 0, B 90, C 0, E1 0, E2 0, E3 0, E4 0} C_DIS
LIN {X -66.52, Y 91.521, Z 42.75, A 0, B 90, C 0, E1 0, E2 0, E3 0, E4 0} C_DIS
LIN {X -65.592, Y 99.567, Z 42.75, A 0, B 90, C 0, E1 0, E2 0, E3 0, E4 0} C_DIS
LIN {X -64.587, Y 107.603, Z 42.75, A 0, B 90, C 0, E1 0, E2 0, E3 0, E4 0} C_DIS
LIN {X -63.507, Y 115.629, Z 42.75, A 0, B 90, C 0, E1 0, E2 0, E3 0, E4 0} C_DIS
LIN {X -62.35, Y 123.645, Z 42.75, A 0, B 90, C 0, E1 0, E2 0, E3 0, E4 0} C_DIS
LIN {X -61.119, Y 131.65, Z 42.75, A 0, B 90, C 0, E1 0, E2 0, E3 0, E4 0} C_DIS
LIN {X -59.813, Y 139.643, Z 42.75, A 0, B 90, C 0, E1 0, E2 0, E3 0, E4 0} C_DIS
LIN {X -58.434, Y 147.623, Z 42.75, A 0, B 90, C 0, E1 0, E2 0, E3 0, E4 0} C_DIS
LIN {X -56.981, Y 155.591, Z 42.75, A 0, B 90, C 0, E1 0, E2 0, E3 0, E4 0} C_DIS
LIN {X -55.456, Y 163.545, Z 42.75, A 0, B 90, C 0, E1 0, E2 0, E3 0, E4 0} C_DIS
LIN {X -53.859, Y 171.485, Z 42.75, A 0, B 90, C 0, E1 0, E2 0, E3 0, E4 0} C_DIS
LIN {X -52.191, Y 179.41, Z 42.75, A 0, B 90, C 0, E1 0, E2 0, E3 0, E4 0} C_DIS
LIN {X -50.453, Y 187.32, Z 42.75, A 0, B 90, C 0, E1 0, E2 0, E3 0, E4 0} C_DIS
LIN {X -48.645, Y 195.215, Z 42.75, A 0, B 90, C 0, E1 0, E2 0, E3 0, E4 0} C_DIS
LIN {X -46.769, Y 203.093, Z 42.75, A 0, B 90, C 0, E1 0, E2 0, E3 0, E4 0} C_DIS
LIN {X -44.824, Y 210.955, Z 42.75, A 0, B 90, C 0, E1 0, E2 0, E3 0, E4 0} C_DIS
LIN {X -42.811, Y 218.8, Z 42.75, A 0, B 90, C 0, E1 0, E2 0, E3 0, E4 0} C_DIS
LIN {X -40.732, Y 226.627, Z 42.75, A 0, B 90, C 0, E1 0, E2 0, E3 0, E4 0} C_DIS
LIN {X -38.586, Y 234.436, Z 42.75, A 0, B 90, C 0, E1 0, E2 0, E3 0, E4 0} C_DIS
LIN {X -36.374, Y 242.228, Z 42.75, A 0, B 90, C 0, E1 0, E2 0, E3 0, E4 0} C_DIS
LIN {X -34.384, Y 250, Z 45.25, A 0, B 90, C 0, E1 0, E2 0, E3 0, E4 0} C_DIS
LIN {X -32.043, Y 257.732, Z 45.25, A 0, B 90, C 0, E1 0, E2 0, E3 0, E4 0} C_DIS
LIN {X -29.639, Y 265.445, Z 45.25, A 0, B 90, C 0, E1 0, E2 0, E3 0, E4 0} C_DIS
LIN {X -27.174, Y 273.139, Z 45.25, A 0, B 90, C 0, E1 0, E2 0, E3 0, E4 0} C_DIS
LIN {X -24.649, Y 280.813, Z 45.25, A 0, B 90, C 0, E1 0, E2 0, E3 0, E4 0} C_DIS
LIN {X -22.064, Y 288.467, Z 45.25, A 0, B 90, C 0, E1 0, E2 0, E3 0, E4 0} C_DIS
LIN {X -19.422, Y 296.102, Z 45.25, A 0, B 90, C 0, E1 0, E2 0, E3 0, E4 0} C_DIS
LIN {X -16.724, Y 303.717, Z 45.25, A 0, B 90, C 0, E1 0, E2 0, E3 0, E4 0} C_DIS
LIN {X -13.97, Y 311.312, Z 45.25, A 0, B 90, C 0, E1 0, E2 0, E3 0, E4 0} C_DIS
LIN {X -11.162, Y 318.887, Z 45.25, A 0, B 90, C 0, E1 0, E2 0, E3 0, E4 0} C_DIS
LIN {X -8.3, Y 326.442, Z 45.25, A 0, B 90, C 0, E1 0, E2 0, E3 0, E4 0} C_DIS
LIN {X -5.383, Y 333.976, Z 45.25, A 0, B 90, C 0, E1 0, E2 0, E3 0, E4 0} C_DIS
LIN {X -2.413, Y 341.489, Z 45.25, A 0, B 90, C 0, E1 0, E2 0, E3 0, E4 0} C_DIS
LIN {X 0.612, Y 348.98, Z 45.25, A 0, B 90, C 0, E1 0, E2 0, E3 0, E4 0} C_DIS
LIN {X 3.691, Y 356.449, Z 45.25, A 0, B 90, C 0, E1 0, E2 0, E3 0, E4 0} C_DIS
LIN {X 6.825, Y 363.896, Z 45.25, A 0, B 90, C 0, E1 0, E2 0, E3 0, E4 0} C_DIS
LIN {X 11.321, Y 370.401, Z 45.25, A 0, B 90, C 0, E1 0, E2 0, E3 0, E4 0} C_DIS
LIN {X 19.103, Y 370.989, Z 45.25, A 0, B 90, C 0, E1 0, E2 0, E3 0, E4 0} C_DIS
LIN {X 26.53, Y 367.81, Z 45.25, A 0, B 90, C 0, E1 0, E2 0, E3 0, E4 0} C_DIS
LIN {X 33.957, Y 364.631, Z 45.25, A 0, B 90, C 0, E1 0, E2 0, E3 0, E4 0} C_DIS
LIN {X 41.384, Y 361.451, Z 45.25, A 0, B 90, C 0, E1 0, E2 0, E3 0, E4 0} C_DIS
LIN {X 48.811, Y 358.272, Z 45.25, A 0, B 90, C 0, E1 0, E2 0, E3 0, E4 0} C_DIS
LIN {X 56.238, Y 355.092, Z 45.25, A 0, B 90, C 0, E1 0, E2 0, E3 0, E4 0} C_DIS
LIN {X 63.665, Y 351.913, Z 45.25, A 0, B 90, C 0, E1 0, E2 0, E3 0, E4 0} C_DIS
LIN {X 70.955, Y 348.467, Z 45.25, A 0, B 90, C 0, E1 0, E2 0, E3 0, E4 0} C_DIS
LIN {X 74.385, Y 341.581, Z 45.25, A 0, B 90, C 0, E1 0, E2 0, E3 0, E4 0} C_DIS
LIN {X 71.463, Y 334.071, Z 45.25, A 0, B 90, C 0, E1 0, E2 0, E3 0, E4 0} C_DIS
LIN {X 68.34, Y 326.62, Z 45.25, A 0, B 90, C 0, E1 0, E2 0, E3 0, E4 0} C_DIS
LIN {X 65.278, Y 319.144, Z 45.25, A 0, B 90, C 0, E1 0, E2 0, E3 0, E4 0} C_DIS
LIN {X 62.276, Y 311.643, Z 45.25, A 0, B 90, C 0, E1 0, E2 0, E3 0, E4 0} C_DIS
LIN {X 59.334, Y 304.119, Z 45.25, A 0, B 90, C 0, E1 0, E2 0, E3 0, E4 0} C_DIS
LIN {X 56.451, Y 296.572, Z 45.25, A 0, B 90, C 0, E1 0, E2 0, E3 0, E4 0} C_DIS
LIN {X 53.628, Y 289.003, Z 45.25, A 0, B 90, C 0, E1 0, E2 0, E3 0, E4 0} C_DIS
LIN {X 50.864, Y 281.412, Z 45.25, A 0, B 90, C 0, E1 0, E2 0, E3 0, E4 0} C_DIS
LIN {X 48.159, Y 273.799, Z 45.25, A 0, B 90, C 0, E1 0, E2 0, E3 0, E4 0} C_DIS
LIN {X 45.513, Y 266.166, Z 45.25, A 0, B 90, C 0, E1 0, E2 0, E3 0, E4 0} C_DIS
LIN {X 42.929, Y 258.511, Z 45.25, A 0, B 90, C 0, E1 0, E2 0, E3 0, E4 0} C_DIS
LIN {X 40.407, Y 250.836, Z 45.25, A 0, B 90, C 0, E1 0, E2 0, E3 0, E4 0} C_DIS
LIN {X 37.949, Y 243.14, Z 45.25, A 0, B 90, C 0, E1 0, E2 0, E3 0, E4 0} C_DIS
LIN {X 35.556, Y 235.424, Z 45.25, A 0, B 90, C 0, E1 0, E2 0, E3 0, E4 0} C_DIS
LIN {X 33.23, Y 227.687, Z 45.25, A 0, B 90, C 0, E1 0, E2 0, E3 0, E4 0} C_DIS
LIN {X 30.972, Y 219.93, Z 45.25, A 0, B 90, C 0, E1 0, E2 0, E3 0, E4 0} C_DIS
LIN {X 28.783, Y 212.153, Z 45.25, A 0, B 90, C 0, E1 0, E2 0, E3 0, E4 0} C_DIS
LIN {X 26.665, Y 204.357, Z 45.25, A 0, B 90, C 0, E1 0, E2 0, E3 0, E4 0} C_DIS
LIN {X 24.619, Y 196.542, Z 45.25, A 0, B 90, C 0, E1 0, E2 0, E3 0, E4 0} C_DIS
LIN {X 22.645, Y 188.708, Z 45.25, A 0, B 90, C 0, E1 0, E2 0, E3 0, E4 0} C_DIS
LIN {X 20.745, Y 180.855, Z 45.25, A 0, B 90, C 0, E1 0, E2 0, E3 0, E4 0} C_DIS
LIN {X 18.92, Y 172.985, Z 45.25, A 0, B 90, C 0, E1 0, E2 0, E3 0, E4 0} C_DIS
LIN {X 17.17, Y 165.098, Z 45.25, A 0, B 90, C 0, E1 0, E2 0, E3 0, E4 0} C_DIS
LIN {X 15.497, Y 157.195, Z 45.25, A 0, B 90, C 0, E1 0, E2 0, E3 0, E4 0} C_DIS
LIN {X 13.901, Y 149.275, Z 45.25, A 0, B 90, C 0, E1 0, E2 0, E3 0, E4 0} C_DIS
LIN {X 12.384, Y 141.34, Z 45.25, A 0, B 90, C 0, E1 0, E2 0, E3 0, E4 0} C_DIS
LIN {X 10.947, Y 133.39, Z 45.25, A 0, B 90, C 0, E1 0, E2 0, E3 0, E4 0} C_DIS
LIN {X 9.589, Y 125.426, Z 45.25, A 0, B 90, C 0, E1 0, E2 0, E3 0, E4 0} C_DIS
LIN {X 8.312, Y 117.449, Z 45.25, A 0, B 90, C 0, E1 0, E2 0, E3 0, E4 0} C_DIS
LIN {X 7.116, Y 109.459, Z 45.25, A 0, B 90, C 0, E1 0, E2 0, E3 0, E4 0} C_DIS
LIN {X 6.001, Y 101.457, Z 45.25, A 0, B 90, C 0, E1 0, E2 0, E3 0, E4 0} C_DIS
LIN {X 4.969, Y 93.444, Z 45.25, A 0, B 90, C 0, E1 0, E2 0, E3 0, E4 0} C_DIS
LIN {X 4.019, Y 85.422, Z 45.25, A 0, B 90, C 0, E1 0, E2 0, E3 0, E4 0} C_DIS
LIN {X 3.153, Y 77.389, Z 45.25, A 0, B 90, C 0, E1 0, E2 0, E3 0, E4 0} C_DIS
LIN {X 2.37, Y 69.349, Z 45.25, A 0, B 90, C 0, E1 0, E2 0, E3 0, E4 0} C_DIS
LIN {X 1.672, Y 61.3, Z 45.25, A 0, B 90, C 0, E1 0, E2 0, E3 0, E4 0} C_DIS
LIN {X 1.058, Y 53.244, Z 45.25, A 0, B 90, C 0, E1 0, E2 0, E3 0, E4 0} C_DIS
LIN {X 0.529, Y 45.183, Z 45.25, A 0, B 90, C 0, E1 0, E2 0, E3 0, E4 0} C_DIS
LIN {X 0.086, Y 37.116, Z 45.25, A 0, B 90, C 0, E1 0, E2 0, E3 0, E4 0} C_DIS
LIN {X -0.271, Y 29.045, Z 45.25, A 0, B 90, C 0, E1 0, E2 0, E3 0, E4 0} C_DIS
LIN {X -0.542, Y 20.971, Z 45.25, A 0, B 90, C 0, E1 0, E2 0, E3 0, E4 0} C_DIS
LIN {X -0.726, Y 12.894, Z 45.25, A 0, B 90, C 0, E1 0, E2 0, E3 0, E4 0} C_DIS
LIN {X -0.824, Y 4.816, Z 45.25, A 0, B 90, C 0, E1 0, E2 0, E3 0, E4 0} C_DIS
LIN {X -0.833, Y -3.263, Z 45.25, A 0, B 90, C 0, E1 0, E2 0, E3 0, E4 0} C_DIS
LIN {X -0.755, Y -11.341, Z 45.25, A 0, B 90, C 0, E1 0, E2 0, E3 0, E4 0} C_DIS
LIN {X -0.59, Y -19.419, Z 45.25, A 0, B 90, C 0, E1 0, E2 0, E3 0, E4 0} C_DIS
LIN {X -0.338, Y -27.494, Z 45.25, A 0, B 90, C 0, E1 0, E2 0, E3 0, E4 0} C_DIS
LIN {X 0.001, Y -35.565, Z 45.25, A 0, B 90, C 0, E1 0, E2 0, E3 0, E4 0} C_DIS
LIN {X 0.426, Y -43.633, Z 45.25, A 0, B 90, C 0, E1 0, E2 0, E3 0, E4 0} C_DIS
LIN {X 0.937, Y -51.696, Z 45.25, A 0, B 90, C 0, E1 0, E2 0, E3 0, E4 0} C_DIS
LIN {X 1.533, Y -59.752, Z 45.25, A 0, B 90, C 0, E1 0, E2 0, E3 0, E4 0} C_DIS
LIN {X 2.215, Y -67.802, Z 45.25, A 0, B 90, C 0, E1 0, E2 0, E3 0, E4 0} C_DIS
LIN {X 2.982, Y -75.845, Z 45.25, A 0, B 90, C 0, E1 0, E2 0, E3 0, E4 0} C_DIS
LIN {X 3.834, Y -83.879, Z 45.25, A 0, B 90, C 0, E1 0, E2 0, E3 0, E4 0} C_DIS
LIN {X 4.769, Y -91.903, Z 45.25, A 0, B 90, C 0, E1 0, E2 0, E3 0, E4 0} C_DIS
LIN {X 5.787, Y -99.918, Z 45.25, A 0, B 90, C 0, E1 0, E2 0, E3 0, E4 0} C_DIS
LIN {X 6.888, Y -107.921, Z 45.25, A 0, B 90, C 0, E1 0, E2 0, E3 0, E4 0} C_DIS
LIN {X 8.071, Y -115.913, Z 45.25, A 0, B 90, C 0, E1 0, E2 0, E3 0, E4 0} C_DIS
LIN {X 9.335, Y -123.892, Z 45.25, A 0, B 90, C 0, E1 0, E2 0, E3 0, E4 0} C_DIS
LIN {X 10.68, Y -131.858, Z 45.25, A 0, B 90, C 0, E1 0, E2 0, E3 0, E4 0} C_DIS
LIN {X 12.105, Y -139.811, Z 45.25, A 0, B 90, C 0, E1 0, E2 0, E3 0, E4 0} C_DIS
LIN {X 13.61, Y -147.748, Z 45.25, A 0, B 90, C 0, E1 0, E2 0, E3 0, E4 0} C_DIS
LIN {X 15.193, Y -155.67, Z 45.25, A 0, B 90, C 0, E1 0, E2 0, E3 0, E4 0} C_DIS
LIN {X 16.853, Y -163.577, Z 45.25, A 0, B 90, C 0, E1 0, E2 0, E3 0, E4 0} C_DIS
LIN {X 18.59, Y -171.467, Z 45.25, A 0, B 90, C 0, E1 0, E2 0, E3 0, E4 0} C_DIS
LIN {X 20.401, Y -179.34, Z 45.25, A 0, B 90, C 0, E1 0, E2 0, E3 0, E4 0} C_DIS
LIN {X 22.287, Y -187.196, Z 45.25, A 0, B 90, C 0, E1 0, E2 0, E3 0, E4 0} C_DIS
LIN {X 24.246, Y -195.033, Z 45.25, A 0, B 90, C 0, E1 0, E2 0, E3 0, E4 0} C_DIS
LIN {X 26.278, Y -202.853, Z 45.25, A 0, B 90, C 0, E1 0, E2 0, E3 0, E4 0} C_DIS
LIN {X 28.379, Y -210.653, Z 45.25, A 0, B 90, C 0, E1 0, E2 0, E3 0, E4 0} C_DIS
LIN {X 30.551, Y -218.435, Z 45.25, A 0, B 90, C 0, E1 0, E2 0, E3 0, E4 0} C_DIS
LIN {X 32.792, Y -226.197, Z 45.25, A 0, B 90, C 0, E1 0, E2 0, E3 0, E4 0} C_DIS
LIN {X 35.1, Y -233.939, Z 45.25, A 0, B 90, C 0, E1 0, E2 0, E3 0, E4 0} C_DIS
LIN {X 37.475, Y -241.661, Z 45.25, A 0, B 90, C 0, E1 0, E2 0, E3 0, E4 0} C_DIS
LIN {X 39.915, Y -249.362, Z 45.25, A 0, B 90, C 0, E1 0, E2 0, E3 0, E4 0} C_DIS
LIN {X 42.42, Y -257.043, Z 45.25, A 0, B 90, C 0, E1 0, E2 0, E3 0, E4 0} C_DIS
LIN {X 44.988, Y -264.703, Z 45.25, A 0, B 90, C 0, E1 0, E2 0, E3 0, E4 0} C_DIS
LIN {X 47.618, Y -272.342, Z 45.25, A 0, B 90, C 0, E1 0, E2 0, E3 0, E4 0} C_DIS
LIN {X 50.309, Y -279.959, Z 45.25, A 0, B 90, C 0, E1 0, E2 0, E3 0, E4 0} C_DIS
LIN {X 53.061, Y -287.555, Z 45.25, A 0, B 90, C 0, E1 0, E2 0, E3 0, E4 0} C_DIS
LIN {X 55.873, Y -295.129, Z 45.25, A 0, B 90, C 0, E1 0, E2 0, E3 0, E4 0} C_DIS
LIN {X 58.746, Y -302.68, Z 45.25, A 0, B 90, C 0, E1 0, E2 0, E3 0, E4 0} C_DIS
LIN {X 61.679, Y -310.207, Z 45.25, A 0, B 90, C 0, E1 0, E2 0, E3 0, E4 0} C_DIS
LIN {X 64.673, Y -317.711, Z 45.25, A 0, B 90, C 0, E1 0, E2 0, E3 0, E4 0} C_DIS
LIN {X 67.728, Y -325.19, Z 45.25, A 0, B 90, C 0, E1 0, E2 0, E3 0, E4 0} C_DIS
LIN {X 70.844, Y -332.643, Z 45.25, A 0, B 90, C 0, E1 0, E2 0, E3 0, E4 0} C_DIS
LIN {X 74.012, Y -340.075, Z 45.25, A 0, B 90, C 0, E1 0, E2 0, E3 0, E4 0} C_DIS
LIN {X 72.141, Y -347.47, Z 45.25, A 0, B 90, C 0, E1 0, E2 0, E3 0, E4 0} C_DIS
LIN {X 65.092, Y -351.305, Z 45.25, A 0, B 90, C 0, E1 0, E2 0, E3 0, E4 0} C_DIS
LIN {X 57.665, Y -354.485, Z 45.25, A 0, B 90, C 0, E1 0, E2 0, E3 0, E4 0} C_DIS
LIN {X 50.238, Y -357.664, Z 45.25, A 0, B 90, C 0, E1 0, E2 0, E3 0, E4 0} C_DIS
LIN {X 42.812, Y -360.843, Z 45.25, A 0, B 90, C 0, E1 0, E2 0, E3 0, E4 0} C_DIS
LIN {X 35.385, Y -364.023, Z 45.25, A 0, B 90, C 0, E1 0, E2 0, E3 0, E4 0} C_DIS
LIN {X 27.958, Y -367.202, Z 45.25, A 0, B 90, C 0, E1 0, E2 0, E3 0, E4 0} C_DIS
LIN {X 20.531, Y -370.382, Z 45.25, A 0, B 90, C 0, E1 0, E2 0, E3 0, E4 0} C_DIS
LIN {X 12.714, Y -371.085, Z 45.25, A 0, B 90, C 0, E1 0, E2 0, E3 0, E4 0} C_DIS
LIN {X 7.433, Y -365.327, Z 45.25, A 0, B 90, C 0, E1 0, E2 0, E3 0, E4 0} C_DIS
LIN {X 4.289, Y -357.885, Z 45.25, A 0, B 90, C 0, E1 0, E2 0, E3 0, E4 0} C_DIS
LIN {X 1.199, Y -350.421, Z 45.25, A 0, B 90, C 0, E1 0, E2 0, E3 0, E4 0} C_DIS
LIN {X -1.836, Y -342.934, Z 45.25, A 0, B 90, C 0, E1 0, E2 0, E3 0, E4 0} C_DIS
LIN {X -4.817, Y -335.425, Z 45.25, A 0, B 90, C 0, E1 0, E2 0, E3 0, E4 0} C_DIS
LIN {X -7.744, Y -327.895, Z 45.25, A 0, B 90, C 0, E1 0, E2 0, E3 0, E4 0} C_DIS
LIN {X -10.617, Y -320.344, Z 45.25, A 0, B 90, C 0, E1 0, E2 0, E3 0, E4 0} C_DIS
LIN {X -13.435, Y -312.773, Z 45.25, A 0, B 90, C 0, E1 0, E2 0, E3 0, E4 0} C_DIS
LIN {X -16.199, Y -305.181, Z 45.25, A 0, B 90, C 0, E1 0, E2 0, E3 0, E4 0} C_DIS
LIN {X -18.908, Y -297.57, Z 45.25, A 0, B 90, C 0, E1 0, E2 0, E3 0, E4 0} C_DIS
LIN {X -21.561, Y -289.939, Z 45.25, A 0, B 90, C 0, E1 0, E2 0, E3 0, E4 0} C_DIS
LIN {X -24.156, Y -282.289, Z 45.25, A 0, B 90, C 0, E1 0, E2 0, E3 0, E4 0} C_DIS
LIN {X -26.692, Y -274.618, Z 45.25, A 0, B 90, C 0, E1 0, E2 0, E3 0, E4 0} C_DIS
LIN {X -29.169, Y -266.928, Z 45.25, A 0, B 90, C 0, E1 0, E2 0, E3 0, E4 0} C_DIS
LIN {X -31.584, Y -259.219, Z 45.25, A 0, B 90, C 0, E1 0, E2 0, E3 0, E4 0} C_DIS
LIN {X -33.937, Y -251.49, Z 45.25, A 0, B 90, C 0, E1 0, E2 0, E3 0, E4 0} C_DIS
LIN {X -36.226, Y -243.742, Z 45.25, A 0, B 90, C 0, E1 0, E2 0, E3 0, E4 0} C_DIS
LIN {X -38.451, Y -235.976, Z 45.25, A 0, B 90, C 0, E1 0, E2 0, E3 0, E4 0} C_DIS
LIN {X -40.611, Y -228.191, Z 45.25, A 0, B 90, C 0, E1 0, E2 0, E3 0, E4 0} C_DIS
LIN {X -42.705, Y -220.388, Z 45.25, A 0, B 90, C 0, E1 0, E2 0, E3 0, E4 0} C_DIS
LIN {X -44.733, Y -212.568, Z 45.25, A 0, B 90, C 0, E1 0, E2 0, E3 0, E4 0} C_DIS
LIN {X -46.693, Y -204.731, Z 45.25, A 0, B 90, C 0, E1 0, E2 0, E3 0, E4 0} C_DIS
LIN {X -48.586, Y -196.877, Z 45.25, A 0, B 90, C 0, E1 0, E2 0, E3 0, E4 0} C_DIS
LIN {X -50.409, Y -189.006, Z 45.25, A 0, B 90, C 0, E1 0, E2 0, E3 0, E4 0} C_DIS
LIN {X -52.163, Y -181.12, Z 45.25, A 0, B 90, C 0, E1 0, E2 0, E3 0, E4 0} C_DIS
LIN {X -53.847, Y -173.219, Z 45.25, A 0, B 90, C 0, E1 0, E2 0, E3 0, E4 0} C_DIS
LIN {X -55.46, Y -165.303, Z 45.25, A 0, B 90, C 0, E1 0, E2 0, E3 0, E4 0} C_DIS
LIN {X -57.002, Y -157.372, Z 45.25, A 0, B 90, C 0, E1 0, E2 0, E3 0, E4 0} C_DIS
LIN {X -58.471, Y -149.428, Z 45.25, A 0, B 90, C 0, E1 0, E2 0, E3 0, E4 0} C_DIS
LIN {X -59.867, Y -141.471, Z 45.25, A 0, B 90, C 0, E1 0, E2 0, E3 0, E4 0} C_DIS
LIN {X -61.189, Y -133.501, Z 45.25, A 0, B 90, C 0, E1 0, E2 0, E3 0, E4 0} C_DIS
LIN {X -62.438, Y -125.519, Z 45.25, A 0, B 90, C 0, E1 0, E2 0, E3 0, E4 0} C_DIS
LIN {X -63.611, Y -117.526, Z 45.25, A 0, B 90, C 0, E1 0, E2 0, E3 0, E4 0} C_DIS
LIN {X -64.709, Y -109.522, Z 45.25, A 0, B 90, C 0, E1 0, E2 0, E3 0, E4 0} C_DIS
LIN {X -65.732, Y -101.508, Z 45.25, A 0, B 90, C 0, E1 0, E2 0, E3 0, E4 0} C_DIS
LIN {X -66.678, Y -93.485, Z 45.25, A 0, B 90, C 0, E1 0, E2 0, E3 0, E4 0} C_DIS
LIN {X -67.549, Y -85.453, Z 45.25, A 0, B 90, C 0, E1 0, E2 0, E3 0, E4 0} C_DIS
LIN {X -68.342, Y -77.413, Z 45.25, A 0, B 90, C 0, E1 0, E2 0, E3 0, E4 0} C_DIS
LIN {X -69.059, Y -69.366, Z 45.25, A 0, B 90, C 0, E1 0, E2 0, E3 0, E4 0} C_DIS
LIN {X -69.698, Y -61.312, Z 45.25, A 0, B 90, C 0, E1 0, E2 0, E3 0, E4 0} C_DIS
LIN {X -70.26, Y -53.253, Z 45.25, A 0, B 90, C 0, E1 0, E2 0, E3 0, E4 0} C_DIS
LIN {X -70.743, Y -45.189, Z 45.25, A 0, B 90, C 0, E1 0, E2 0, E3 0, E4 0} C_DIS
LIN {X -71.148, Y -37.12, Z 45.25, A 0, B 90, C 0, E1 0, E2 0, E3 0, E4 0} C_DIS
LIN {X -71.475, Y -29.048, Z 45.25, A 0, B 90, C 0, E1 0, E2 0, E3 0, E4 0} C_DIS
LIN {X -71.722, Y -20.973, Z 45.25, A 0, B 90, C 0, E1 0, E2 0, E3 0, E4 0} C_DIS
LIN {X -71.89, Y -12.896, Z 45.25, A 0, B 90, C 0, E1 0, E2 0, E3 0, E4 0} C_DIS
LIN {X -71.978, Y -4.817, Z 45.25, A 0, B 90, C 0, E1 0, E2 0, E3 0, E4 0} C_DIS
LIN {X -71.986, Y 3.262, Z 45.25, A 0, B 90, C 0, E1 0, E2 0, E3 0, E4 0} C_DIS
LIN {X -71.914, Y 11.34, Z 45.25, A 0, B 90, C 0, E1 0, E2 0, E3 0, E4 0} C_DIS
LIN {X -71.762, Y 19.418, Z 45.25, A 0, B 90, C 0, E1 0, E2 0, E3 0, E4 0} C_DIS
LIN {X -71.531, Y 27.493, Z 45.25, A 0, B 90, C 0, E1 0, E2 0, E3 0, E4 0} C_DIS
LIN {X -71.22, Y 35.566, Z 45.25, A 0, B 90, C 0, E1 0, E2 0, E3 0, E4 0} C_DIS
LIN {X -70.831, Y 43.636, Z 45.25, A 0, B 90, C 0, E1 0, E2 0, E3 0, E4 0} C_DIS
LIN {X -70.363, Y 51.701, Z 45.25, A 0, B 90, C 0, E1 0, E2 0, E3 0, E4 0} C_DIS
LIN {X -69.817, Y 59.761, Z 45.25, A 0, B 90, C 0, E1 0, E2 0, E3 0, E4 0} C_DIS
LIN {X -69.192, Y 67.816, Z 45.25, A 0, B 90, C 0, E1 0, E2 0, E3 0, E4 0} C_DIS
LIN {X -68.491, Y 75.864, Z 45.25, A 0, B 90, C 0, E1 0, E2 0, E3 0, E4 0} C_DIS
LIN {X -67.711, Y 83.905, Z 45.25, A 0, B 90, C 0, E1 0, E2 0, E3 0, E4 0} C_DIS
LIN {X -66.855, Y 91.939, Z 45.25, A 0, B 90, C 0, E1 0, E2 0, E3 0, E4 0} C_DIS
LIN {X -65.923, Y 99.964, Z 45.25, A 0, B 90, C 0, E1 0, E2 0, E3 0, E4 0} C_DIS
LIN {X -64.914, Y 107.979, Z 45.25, A 0, B 90, C 0, E1 0, E2 0, E3 0, E4 0} C_DIS
LIN {X -63.829, Y 115.985, Z 45.25, A 0, B 90, C 0, E1 0, E2 0, E3 0, E4 0} C_DIS
LIN {X -62.669, Y 123.98, Z 45.25, A 0, B 90, C 0, E1 0, E2 0, E3 0, E4 0} C_DIS
LIN {X -61.434, Y 131.964, Z 45.25, A 0, B 90, C 0, E1 0, E2 0, E3 0, E4 0} C_DIS
LIN {X -60.125, Y 139.936, Z 45.25, A 0, B 90, C 0, E1 0, E2 0, E3 0, E4 0} C_DIS
LIN {X -58.742, Y 147.896, Z 45.25, A 0, B 90, C 0, E1 0, E2 0, E3 0, E4 0} C_DIS
LIN {X -57.287, Y 155.843, Z 45.25, A 0, B 90, C 0, E1 0, E2 0, E3 0, E4 0} C_DIS
LIN {X -55.759, Y 163.776, Z 45.25, A 0, B 90, C 0, E1 0, E2 0, E3 0, E4 0} C_DIS
LIN {X -54.16, Y 171.695, Z 45.25, A 0, B 90, C 0, E1 0, E2 0, E3 0, E4 0} C_DIS
LIN {X -52.489, Y 179.599, Z 45.25, A 0, B 90, C 0, E1 0, E2 0, E3 0, E4 0} C_DIS
LIN {X -50.749, Y 187.488, Z 45.25, A 0, B 90, C 0, E1 0, E2 0, E3 0, E4 0} C_DIS
LIN {X -48.939, Y 195.362, Z 45.25, A 0, B 90, C 0, E1 0, E2 0, E3 0, E4 0} C_DIS
LIN {X -47.061, Y 203.219, Z 45.25, A 0, B 90, C 0, E1 0, E2 0, E3 0, E4 0} C_DIS
LIN {X -45.114, Y 211.06, Z 45.25, A 0, B 90, C 0, E1 0, E2 0, E3 0, E4 0} C_DIS
LIN {X -43.1, Y 218.884, Z 45.25, A 0, B 90, C 0, E1 0, E2 0, E3 0, E4 0} C_DIS
LIN {X -41.019, Y 226.69, Z 45.25, A 0, B 90, C 0, E1 0, E2 0, E3 0, E4 0} C_DIS
LIN {X -38.873, Y 234.479, Z 45.25, A 0, B 90, C 0, E1 0, E2 0, E3 0, E4 0} C_DIS
LIN {X -36.66, Y 242.249, Z 45.25, A 0, B 90, C 0, E1 0, E2 0, E3 0, E4 0} C_DIS
LIN {X -34.668, Y 250, Z 47.75, A 0, B 90, C 0, E1 0, E2 0, E3 0, E4 0} C_DIS
LIN {X -32.327, Y 257.711, Z 47.75, A 0, B 90, C 0, E1 0, E2 0, E3 0, E4 0} C_DIS
LIN {X -29.923, Y 265.403, Z 47.75, A 0, B 90, C 0, E1 0, E2 0, E3 0, E4 0} C_DIS
LIN {X -27.458, Y 273.076, Z 47.75, A 0, B 90, C 0, E1 0, E2 0, E3 0, E4 0} C_DIS
LIN {X -24.932, Y 280.729, Z 47.75, A 0, B 90, C 0, E1 0, E2 0, E3 0, E4 0} C_DIS
LIN {X -22.348, Y 288.362, Z 47.75, A 0, B 90, C 0, E1 0, E2 0, E3 0, E4 0} C_DIS
LIN {X -19.706, Y 295.976, Z 47.75, A 0, B 90, C 0, E1 0, E2 0, E3 0, E4 0} C_DIS
LIN {X -17.008, Y 303.57, Z 47.75, A 0, B 90, C 0, E1 0, E2 0, E3 0, E4 0} C_DIS
LIN {X -14.255, Y 311.144, Z 47.75, A 0, B 90, C 0, E1 0, E2 0, E3 0, E4 0} C_DIS
LIN {X -11.449, Y 318.698, Z 47.75, A 0, B 90, C 0, E1 0, E2 0, E3 0, E4 0} C_DIS
LIN {X -8.588, Y 326.232, Z 47.75, A 0, B 90, C 0, E1 0, E2 0, E3 0, E4 0} C_DIS
LIN {X -5.674, Y 333.746, Z 47.75, A 0, B 90, C 0, E1 0, E2 0, E3 0, E4 0} C_DIS
LIN {X -2.705, Y 341.238, Z 47.75, A 0, B 90, C 0, E1 0, E2 0, E3 0, E4 0} C_DIS
LIN {X 0.318, Y 348.708, Z 47.75, A 0, B 90, C 0, E1 0, E2 0, E3 0, E4 0} C_DIS
LIN {X 3.395, Y 356.157, Z 47.75, A 0, B 90, C 0, E1 0, E2 0, E3 0, E4 0} C_DIS
LIN {X 6.527, Y 363.582, Z 47.75, A 0, B 90, C 0, E1 0, E2 0, E3 0, E4 0} C_DIS
LIN {X 11.113, Y 369.984, Z 47.75, A 0, B 90, C 0, E1 0, E2 0, E3 0, E4 0} C_DIS
LIN {X 18.891, Y 370.407, Z 47.75, A 0, B 90, C 0, E1 0, E2 0, E3 0, E4 0} C_DIS
LIN {X 26.299, Y 367.234, Z 47.75, A 0, B 90, C 0, E1 0, E2 0, E3 0, E4 0} C_DIS
LIN {X 33.707, Y 364.061, Z 47.75, A 0, B 90, C 0, E1 0, E2 0, E3 0, E4 0} C_DIS
LIN {X 41.115, Y 360.887, Z 47.75, A 0, B 90, C 0, E1 0, E2 0, E3 0, E4 0} C_DIS
LIN {X 48.522, Y 357.714, Z 47.75, A 0, B 90, C 0, E1 0, E2 0, E3 0, E4 0} C_DIS
LIN {X 55.93, Y 354.541, Z 47.75, A 0, B 90, C 0, E1 0, E2 0, E3 0, E4 0} C_DIS
LIN {X 63.338, Y 351.368, Z 47.75, A 0, B 90, C 0, E1 0, E2 0, E3 0, E4 0} C_DIS
LIN {X 70.334, Y 347.489, Z 47.75, A 0, B 90, C 0, E1 0, E2 0, E3 0, E4 0} C_DIS
LIN {X 72.055, Y 340.08, Z 47.75, A 0, B 90, C 0, E1 0, E2 0, E3 0, E4 0} C_DIS
LIN {X 68.892, Y 332.668, Z 47.75, A 0, B 90, C 0, E1 0, E2 0, E3 0, E4 0} C_DIS
LIN {X 65.785, Y 325.232, Z 47.75, A 0, B 90, C 0, E1 0, E2 0, E3 0, E4 0} C_DIS
LIN {X 62.738, Y 317.771, Z 47.75, A 0, B 90, C 0, E1 0, E2 0, E3 0, E4 0} C_DIS
LIN {X 59.751, Y 310.286, Z 47.75, A 0, B 90, C 0, E1 0, E2 0, E3 0, E4 0} C_DIS
LIN {X 56.823, Y 302.778, Z 47.75, A 0, B 90, C 0, E1 0, E2 0, E3 0, E4 0} C_DIS
LIN {X 53.955, Y 295.247, Z 47.75, A 0, B 90, C 0, E1 0, E2 0, E3 0, E4 0} C_DIS
LIN {X 51.146, Y 287.693, Z 47.75, A 0, B 90, C 0, E1 0, E2 0, E3 0, E4 0} C_DIS
LIN {X 48.396, Y 280.118, Z 47.75, A 0, B 90, C 0, E1 0, E2 0, E3 0, E4 0} C_DIS
LIN {X 45.704, Y 272.522, Z 47.75, A 0, B 90, C 0, E1 0, E2 0, E3 0, E4 0} C_DIS
LIN {X 43.072, Y 264.905, Z 47.75, A 0, B 90, C 0, E1 0, E2 0, E3 0, E4 0} C_DIS
LIN {X 40.502, Y 257.267, Z 47.75, A 0, B 90, C 0, E1 0, E2 0, E3 0, E4 0} C_DIS
LIN {X 37.994, Y 249.608, Z 47.75, A 0, B 90, C 0, E1 0, E2 0, E3 0, E4 0} C_DIS
LIN {X 35.549, Y 241.929, Z 47.75, A 0, B 90, C 0, E1 0, E2 0, E3 0, E4 0} C_DIS
LIN {X 33.17, Y 234.229, Z 47.75, A 0, B 90, C 0, E1 0, E2 0, E3 0, E4 0} C_DIS
LIN {X 30.857, Y 226.509, Z 47.75, A 0, B 90, C 0, E1 0, E2 0, E3 0, E4 0} C_DIS
LIN {X 28.613, Y 218.769, Z 47.75, A 0, B 90, C 0, E1 0, E2 0, E3 0, E4 0} C_DIS
LIN {X 26.437, Y 211.01, Z 47.75, A 0, B 90, C 0, E1 0, E2 0, E3 0, E4 0} C_DIS
LIN {X 24.332, Y 203.231, Z 47.75, A 0, B 90, C 0, E1 0, E2 0, E3 0, E4 0} C_DIS
LIN {X 22.299, Y 195.432, Z 47.75, A 0, B 90, C 0, E1 0, E2 0, E3 0, E4 0} C_DIS
LIN {X 20.338, Y 187.616, Z 47.75, A 0, B 90, C 0, E1 0, E2 0, E3 0, E4 0} C_DIS
LIN {X 18.451, Y 179.781, Z 47.75, A 0, B 90, C 0, E1 0, E2 0, E3 0, E4 0} C_DIS
LIN {X 16.639, Y 171.928, Z 47.75, A 0, B 90, C 0, E1 0, E2 0, E3 0, E4 0} C_DIS
LIN {X 14.901, Y 164.059, Z 47.75, A 0, B 90, C 0, E1 0, E2 0, E3 0, E4 0} C_DIS
LIN {X 13.24, Y 156.173, Z 47.75, A 0, B 90, C 0, E1 0, E2 0, E3 0, E4 0} C_DIS
LIN {X 11.657, Y 148.271, Z 47.75, A 0, B 90, C 0, E1 0, E2 0, E3 0, E4 0} C_DIS
LIN {X 10.152, Y 140.354, Z 47.75, A 0, B 90, C 0, E1 0, E2 0, E3 0, E4 0} C_DIS
LIN {X 8.726, Y 132.422, Z 47.75, A 0, B 90, C 0, E1 0, E2 0, E3 0, E4 0} C_DIS
LIN {X 7.38, Y 124.477, Z 47.75, A 0, B 90, C 0, E1 0, E2 0, E3 0, E4 0} C_DIS
LIN {X 6.114, Y 116.518, Z 47.75, A 0, B 90, C 0, E1 0, E2 0, E3 0, E4 0} C_DIS
LIN {X 4.929, Y 108.547, Z 47.75, A 0, B 90, C 0, E1 0, E2 0, E3 0, E4 0} C_DIS
LIN {X 3.826, Y 100.564, Z 47.75, A 0, B 90, C 0, E1 0, E2 0, E3 0, E4 0} C_DIS
LIN {X 2.804, Y 92.57, Z 47.75, A 0, B 90, C 0, E1 0, E2 0, E3 0, E4 0} C_DIS
LIN {X 1.865, Y 84.566, Z 47.75, A 0, B 90, C 0, E1 0, E2 0, E3 0, E4 0} C_DIS
LIN {X 1.008, Y 76.553, Z 47.75, A 0, B 90, C 0, E1 0, E2 0, E3 0, E4 0} C_DIS
LIN {X 0.235, Y 68.531, Z 47.75, A 0, B 90, C 0, E1 0, E2 0, E3 0, E4 0} C_DIS
LIN {X -0.453, Y 60.502, Z 47.75, A 0, B 90, C 0, E1 0, E2 0, E3 0, E4 0} C_DIS
LIN {X -1.058, Y 52.465, Z 47.75, A 0, B 90, C 0, E1 0, E2 0, E3 0, E4 0} C_DIS
LIN {X -1.578, Y 44.423, Z 47.75, A 0, B 90, C 0, E1 0, E2 0, E3 0, E4 0} C_DIS
LIN {X -2.012, Y 36.376, Z 47.75, A 0, B 90, C 0, E1 0, E2 0, E3 0, E4 0} C_DIS
LIN {X -2.361, Y 28.325, Z 47.75, A 0, B 90, C 0, E1 0, E2 0, E3 0, E4 0} C_DIS
LIN {X -2.624, Y 20.27, Z 47.75, A 0, B 90, C 0, E1 0, E2 0, E3 0, E4 0} C_DIS
LIN {X -2.801, Y 12.213, Z 47.75, A 0, B 90, C 0, E1 0, E2 0, E3 0, E4 0} C_DIS
LIN {X -2.891, Y 4.155, Z 47.75, A 0, B 90, C 0, E1 0, E2 0, E3 0, E4 0} C_DIS
LIN {X -2.894, Y -3.904, Z 47.75, A 0, B 90, C 0, E1 0, E2 0, E3 0, E4 0} C_DIS
LIN {X -2.809, Y -11.962, Z 47.75, A 0, B 90, C 0, E1 0, E2 0, E3 0, E4 0} C_DIS
LIN {X -2.638, Y -20.02, Z 47.75, A 0, B 90, C 0, E1 0, E2 0, E3 0, E4 0} C_DIS
LIN {X -2.38, Y -28.074, Z 47.75, A 0, B 90, C 0, E1 0, E2 0, E3 0, E4 0} C_DIS
LIN {X -2.036, Y -36.126, Z 47.75, A 0, B 90, C 0, E1 0, E2 0, E3 0, E4 0} C_DIS
LIN {X -1.605, Y -44.173, Z 47.75, A 0, B 90, C 0, E1 0, E2 0, E3 0, E4 0} C_DIS
LIN {X -1.09, Y -52.216, Z 47.75, A 0, B 90, C 0, E1 0, E2 0, E3 0, E4 0} C_DIS
LIN {X -0.488, Y -60.252, Z 47.75, A 0, B 90, C 0, E1 0, E2 0, E3 0, E4 0} C_DIS
LIN {X 0.198, Y -68.282, Z 47.75, A 0, B 90, C 0, E1 0, E2 0, E3 0, E4 0} C_DIS
LIN {X 0.968, Y -76.304, Z 47.75, A 0, B 90, C 0, E1 0, E2 0, E3 0, E4 0} C_DIS
LIN {X 1.823, Y -84.317, Z 47.75, A 0, B 90, C 0, E1 0, E2 0, E3 0, E4 0} C_DIS
LIN {X 2.762, Y -92.321, Z 47.75, A 0, B 90, C 0, E1 0, E2 0, E3 0, E4 0} C_DIS
LIN {X 3.783, Y -100.315, Z 47.75, A 0, B 90, C 0, E1 0, E2 0, E3 0, E4 0} C_DIS
LIN {X 4.886, Y -108.298, Z 47.75, A 0, B 90, C 0, E1 0, E2 0, E3 0, E4 0} C_DIS
LIN {X 6.072, Y -116.269, Z 47.75, A 0, B 90, C 0, E1 0, E2 0, E3 0, E4 0} C_DIS
LIN {X 7.338, Y -124.228, Z 47.75, A 0, B 90, C 0, E1 0, E2 0, E3 0, E4 0} C_DIS
LIN {X 8.684, Y -132.174, Z 47.75, A 0, B 90, C 0, E1 0, E2 0, E3 0, E4 0} C_DIS
LIN {X 10.11, Y -140.105, Z 47.75, A 0, B 90, C 0, E1 0, E2 0, E3 0, E4 0} C_DIS
LIN {X 11.616, Y -148.022, Z 47.75, A 0, B 90, C 0, E1 0, E2 0, E3 0, E4 0} C_DIS
LIN {X 13.199, Y -155.924, Z 47.75, A 0, B 90, C 0, E1 0, E2 0, E3 0, E4 0} C_DIS
LIN {X 14.86, Y -163.81, Z 47.75, A 0, B 90, C 0, E1 0, E2 0, E3 0, E4 0} C_DIS
LIN {X 16.596, Y -171.68, Z 47.75, A 0, B 90, C 0, E1 0, E2 0, E3 0, E4 0} C_DIS
LIN {X 18.408, Y -179.532, Z 47.75, A 0, B 90, C 0, E1 0, E2 0, E3 0, E4 0} C_DIS
LIN {X 20.293, Y -187.368, Z 47.75, A 0, B 90, C 0, E1 0, E2 0, E3 0, E4 0} C_DIS
LIN {X 22.251, Y -195.185, Z 47.75, A 0, B 90, C 0, E1 0, E2 0, E3 0, E4 0} C_DIS
LIN {X 24.28, Y -202.984, Z 47.75, A 0, B 90, C 0, E1 0, E2 0, E3 0, E4 0} C_DIS
LIN {X 26.38, Y -210.765, Z 47.75, A 0, B 90, C 0, E1 0, E2 0, E3 0, E4 0} C_DIS
LIN {X 28.55, Y -218.526, Z 47.75, A 0, B 90, C 0, E1 0, E2 0, E3 0, E4 0} C_DIS
LIN {X 30.788, Y -226.268, Z 47.75, A 0, B 90, C 0, E1 0, E2 0, E3 0, E4 0} C_DIS
LIN {X 33.093, Y -233.99, Z 47.75, A 0, B 90, C 0, E1 0, E2 0, E3 0, E4 0} C_DIS
LIN {X 35.465, Y -241.692, Z 47.75, A 0, B 90, C 0, E1 0, E2 0, E3 0, E4 0} C_DIS
LIN {X 37.901, Y -249.374, Z 47.75, A 0, B 90, C 0, E1 0, E2 0, E3 0, E4 0} C_DIS
LIN {X 40.402, Y -257.035, Z 47.75, A 0, B 90, C 0, E1 0, E2 0, E3 0, E4 0} C_DIS
LIN {X 42.966, Y -264.675, Z 47.75, A 0, B 90, C 0, E1 0, E2 0, E3 0, E4 0} C_DIS
LIN {X 45.592, Y -272.294, Z 47.75, A 0, B 90, C 0, E1 0, E2 0, E3 0, E4 0} C_DIS
LIN {X 48.279, Y -279.892, Z 47.75, A 0, B 90, C 0, E1 0, E2 0, E3 0, E4 0} C_DIS
LIN {X 51.026, Y -287.468, Z 47.75, A 0, B 90, C 0, E1 0, E2 0, E3 0, E4 0} C_DIS
LIN {X 53.834, Y -295.022, Z 47.75, A 0, B 90, C 0, E1 0, E2 0, E3 0, E4 0} C_DIS
LIN {X 56.702, Y -302.553, Z 47.75, A 0, B 90, C 0, E1 0, E2 0, E3 0, E4 0} C_DIS
LIN {X 59.63, Y -310.061, Z 47.75, A 0, B 90, C 0, E1 0, E2 0, E3 0, E4 0} C_DIS
LIN {X 62.619, Y -317.545, Z 47.75, A 0, B 90, C 0, E1 0, E2 0, E3 0, E4 0} C_DIS
LIN {X 65.669, Y -325.005, Z 47.75, A 0, B 90, C 0, E1 0, E2 0, E3 0, E4 0} C_DIS
LIN {X 68.779, Y -332.439, Z 47.75, A 0, B 90, C 0, E1 0, E2 0, E3 0, E4 0} C_DIS
LIN {X 71.951, Y -339.848, Z 47.75, A 0, B 90, C 0, E1 0, E2 0, E3 0, E4 0} C_DIS
LIN {X 70.504, Y -347.308, Z 47.75, A 0, B 90, C 0, E1 0, E2 0, E3 0, E4 0} C_DIS
LIN {X 63.568, Y -351.273, Z 47.75, A 0, B 90, C 0, E1 0, E2 0, E3 0, E4 0} C_DIS
LIN {X 56.161, Y -354.446, Z 47.75, A 0, B 90, C 0, E1 0, E2 0, E3 0, E4 0} C_DIS
LIN {X 48.753, Y -357.619, Z 47.75, A 0, B 90, C 0, E1 0, E2 0, E3 0, E4 0} C_DIS
LIN {X 41.345, Y -360.792, Z 47.75, A 0, B 90, C 0, E1 0, E2 0, E3 0, E4 0} C_DIS
LIN {X 33.937, Y -363.965, Z 47.75, A 0, B 90, C 0, E1 0, E2 0, E3 0, E4 0} C_DIS
LIN {X 26.529, Y -367.139, Z 47.75, A 0, B 90, C 0, E1 0, E2 0, E3 0, E4 0} C_DIS
LIN {X 19.121, Y -370.312, Z 47.75, A 0, B 90, C 0, E1 0, E2 0, E3 0, E4 0} C_DIS
LIN {X 11.332, Y -370.109, Z 47.75, A 0, B 90, C 0, E1 0, E2 0, E3 0, E4 0} C_DIS
LIN {X 6.625, Y -363.816, Z 47.75, A 0, B 90, C 0, E1 0, E2 0, E3 0, E4 0} C_DIS
LIN {X 3.491, Y -356.391, Z 47.75, A 0, B 90, C 0, E1 0, E2 0, E3 0, E4 0} C_DIS
LIN {X 0.412, Y -348.943, Z 47.75, A 0, B 90, C 0, E1 0, E2 0, E3 0, E4 0} C_DIS
LIN {X -2.613, Y -341.474, Z 47.75, A 0, B 90, C 0, E1 0, E2 0, E3 0, E4 0} C_DIS
LIN {X -5.583, Y -333.982, Z 47.75, A 0, B 90, C 0, E1 0, E2 0, E3 0, E4 0} C_DIS
LIN {X -8.5, Y -326.47, Z 47.75, A 0, B 90, C 0, E1 0, E2 0, E3 0, E4 0} C_DIS
LIN {X -11.362, Y -318.936, Z 47.75, A 0, B 90, C 0, E1 0, E2 0, E3 0, E4 0} C_DIS
LIN {X -14.17, Y -311.382, Z 47.75, A 0, B 90, C 0, E1 0, E2 0, E3 0, E4 0} C_DIS
LIN {X -16.924, Y -303.809, Z 47.75, A 0, B 90, C 0, E1 0, E2 0, E3 0, E4 0} C_DIS
LIN {X -19.623, Y -296.215, Z 47.75, A 0, B 90, C 0, E1 0, E2 0, E3 0, E4 0} C_DIS
LIN {X -22.266, Y -288.602, Z 47.75, A 0, B 90, C 0, E1 0, E2 0, E3 0, E4 0} C_DIS
LIN {X -24.852, Y -280.969, Z 47.75, A 0, B 90, C 0, E1 0, E2 0, E3 0, E4 0} C_DIS
LIN {X -27.379, Y -273.317, Z 47.75, A 0, B 90, C 0, E1 0, E2 0, E3 0, E4 0} C_DIS
LIN {X -29.845, Y -265.645, Z 47.75, A 0, B 90, C 0, E1 0, E2 0, E3 0, E4 0} C_DIS
LIN {X -32.251, Y -257.953, Z 47.75, A 0, B 90, C 0, E1 0, E2 0, E3 0, E4 0} C_DIS
LIN {X -34.594, Y -250.242, Z 47.75, A 0, B 90, C 0, E1 0, E2 0, E3 0, E4 0} C_DIS
LIN {X -36.874, Y -242.513, Z 47.75, A 0, B 90, C 0, E1 0, E2 0, E3 0, E4 0} C_DIS
LIN {X -39.09, Y -234.764, Z 47.75, A 0, B 90, C 0, E1 0, E2 0, E3 0, E4 0} C_DIS
LIN {X -41.24, Y -226.998, Z 47.75, A 0, B 90, C 0, E1 0, E2 0, E3 0, E4 0} C_DIS
LIN {X -43.325, Y -219.213, Z 47.75, A 0, B 90, C 0, E1 0, E2 0, E3 0, E4 0} C_DIS
LIN {X -45.344, Y -211.411, Z 47.75, A 0, B 90, C 0, E1 0, E2 0, E3 0, E4 0} C_DIS
LIN {X -47.295, Y -203.592, Z 47.75, A 0, B 90, C 0, E1 0, E2 0, E3 0, E4 0} C_DIS
LIN {X -49.178, Y -195.756, Z 47.75, A 0, B 90, C 0, E1 0, E2 0, E3 0, E4 0} C_DIS
LIN {X -50.992, Y -187.904, Z 47.75, A 0, B 90, C 0, E1 0, E2 0, E3 0, E4 0} C_DIS
LIN {X -52.737, Y -180.036, Z 47.75, A 0, B 90, C 0, E1 0, E2 0, E3 0, E4 0} C_DIS
LIN {X -54.412, Y -172.154, Z 47.75, A 0, B 90, C 0, E1 0, E2 0, E3 0, E4 0} C_DIS
LIN {X -56.016, Y -164.256, Z 47.75, A 0, B 90, C 0, E1 0, E2 0, E3 0, E4 0} C_DIS
LIN {X -57.549, Y -156.344, Z 47.75, A 0, B 90, C 0, E1 0, E2 0, E3 0, E4 0} C_DIS
LIN {X -59.009, Y -148.419, Z 47.75, A 0, B 90, C 0, E1 0, E2 0, E3 0, E4 0} C_DIS
LIN {X -60.396, Y -140.48, Z 47.75, A 0, B 90, C 0, E1 0, E2 0, E3 0, E4 0} C_DIS
LIN {X -61.71, Y -132.529, Z 47.75, A 0, B 90, C 0, E1 0, E2 0, E3 0, E4 0} C_DIS
LIN {X -62.95, Y -124.566, Z 47.75, A 0, B 90, C 0, E1 0, E2 0, E3 0, E4 0} C_DIS
LIN {X -64.115, Y -116.592, Z 47.75, A 0, B 90, C 0, E1 0, E2 0, E3 0, E4 0} C_DIS
LIN {X -65.205, Y -108.607, Z 47.75, A 0, B 90, C 0, E1 0, E2 0, E3 0, E4 0} C_DIS
LIN {X -66.219, Y -100.612, Z 47.75, A 0, B 90, C 0, E1 0, E2 0, E3 0, E4 0} C_DIS
LIN {X -67.158, Y -92.608, Z 47.75, A 0, B 90, C 0, E1 0, E2 0, E3 0, E4 0} C_DIS
LIN {X -68.021, Y -84.595, Z 47.75, A 0, B 90, C 0, E1 0, E2 0, E3 0, E4 0} C_DIS
LIN {X -68.807, Y -76.575, Z 47.75, A 0, B 90, C 0, E1 0, E2 0, E3 0, E4 0} C_DIS
LIN {X -69.516, Y -68.547, Z 47.75, A 0, B 90, C 0, E1 0, E2 0, E3 0, E4 0} C_DIS
LIN {X -70.148, Y -60.513, Z 47.75, A 0, B 90, C 0, E1 0, E2 0, E3 0, E4 0} C_DIS
LIN {X -70.702, Y -52.473, Z 47.75, A 0, B 90, C 0, E1 0, E2 0, E3 0, E4 0} C_DIS
LIN {X -71.178, Y -44.429, Z 47.75, A 0, B 90, C 0, E1 0, E2 0, E3 0, E4 0} C_DIS
LIN {X -71.576, Y -36.38, Z 47.75, A 0, B 90, C 0, E1 0, E2 0, E3 0, E4 0} C_DIS
LIN {X -71.896, Y -28.327, Z 47.75, A 0, B 90, C 0, E1 0, E2 0, E3 0, E4 0} C_DIS
LIN {X -72.137, Y -20.272, Z 47.75, A 0, B 90, C 0, E1 0, E2 0, E3 0, E4 0} C_DIS
LIN {X -72.298, Y -12.215, Z 47.75, A 0, B 90, C 0, E1 0, E2 0, E3 0, E4 0} C_DIS
LIN {X -72.38, Y -4.156, Z 47.75, A 0, B 90, C 0, E1 0, E2 0, E3 0, E4 0} C_DIS
LIN {X -72.381, Y 3.903, Z 47.75, A 0, B 90, C 0, E1 0, E2 0, E3 0, E4 0} C_DIS
LIN {X -72.303, Y 11.961, Z 47.75, A 0, B 90, C 0, E1 0, E2 0, E3 0, E4 0} C_DIS
LIN {X -72.145, Y 20.019, Z 47.75, A 0, B 90, C 0, E1 0, E2 0, E3 0, E4 0} C_DIS
LIN {X -71.907, Y 28.074, Z 47.75, A 0, B 90, C 0, E1 0, E2 0, E3 0, E4 0} C_DIS
LIN {X -71.591, Y 36.127, Z 47.75, A 0, B 90, C 0, E1 0, E2 0, E3 0, E4 0} C_DIS
LIN {X -71.196, Y 44.176, Z 47.75, A 0, B 90, C 0, E1 0, E2 0, E3 0, E4 0} C_DIS
LIN {X -70.722, Y 52.221, Z 47.75, A 0, B 90, C 0, E1 0, E2 0, E3 0, E4 0} C_DIS
LIN {X -70.171, Y 60.261, Z 47.75, A 0, B 90, C 0, E1 0, E2 0, E3 0, E4 0} C_DIS
LIN {X -69.541, Y 68.295, Z 47.75, A 0, B 90, C 0, E1 0, E2 0, E3 0, E4 0} C_DIS
LIN {X -68.835, Y 76.323, Z 47.75, A 0, B 90, C 0, E1 0, E2 0, E3 0, E4 0} C_DIS
LIN {X -68.051, Y 84.344, Z 47.75, A 0, B 90, C 0, E1 0, E2 0, E3 0, E4 0} C_DIS
LIN {X -67.19, Y 92.356, Z 47.75, A 0, B 90, C 0, E1 0, E2 0, E3 0, E4 0} C_DIS
LIN {X -66.253, Y 100.361, Z 47.75, A 0, B 90, C 0, E1 0, E2 0, E3 0, E4 0} C_DIS
LIN {X -65.24, Y 108.356, Z 47.75, A 0, B 90, C 0, E1 0, E2 0, E3 0, E4 0} C_DIS
LIN {X -64.151, Y 116.341, Z 47.75, A 0, B 90, C 0, E1 0, E2 0, E3 0, E4 0} C_DIS
LIN {X -62.987, Y 124.315, Z 47.75, A 0, B 90, C 0, E1 0, E2 0, E3 0, E4 0} C_DIS
LIN {X -61.749, Y 132.278, Z 47.75, A 0, B 90, C 0, E1 0, E2 0, E3 0, E4 0} C_DIS
LIN {X -60.436, Y 140.23, Z 47.75, A 0, B 90, C 0, E1 0, E2 0, E3 0, E4 0} C_DIS
LIN {X -59.05, Y 148.168, Z 47.75, A 0, B 90, C 0, E1 0, E2 0, E3 0, E4 0} C_DIS
LIN {X -57.592, Y 156.094, Z 47.75, A 0, B 90, C 0, E1 0, E2 0, E3 0, E4 0} C_DIS
LIN {X -56.061, Y 164.006, Z 47.75, A 0, B 90, C 0, E1 0, E2 0, E3 0, E4 0} C_DIS
LIN {X -54.46, Y 171.904, Z 47.75, A 0, B 90, C 0, E1 0, E2 0, E3 0, E4 0} C_DIS
LIN {X -52.787, Y 179.788, Z 47.75, A 0, B 90, C 0, E1 0, E2 0, E3 0, E4 0} C_DIS
LIN {X -51.045, Y 187.656, Z 47.75, A 0, B 90, C 0, E1 0, E2 0, E3 0, E4 0} C_DIS
LIN {X -49.233, Y 195.509, Z 47.75, A 0, B 90, C 0, E1 0, E2 0, E3 0, E4 0} C_DIS
LIN {X -47.353, Y 203.345, Z 47.75, A 0, B 90, C 0, E1 0, E2 0, E3 0, E4 0} C_DIS
LIN {X -45.404, Y 211.165, Z 47.75, A 0, B 90, C 0, E1 0, E2 0, E3 0, E4 0} C_DIS
LIN {X -43.389, Y 218.968, Z 47.75, A 0, B 90, C 0, E1 0, E2 0, E3 0, E4 0} C_DIS
LIN {X -41.307, Y 226.753, Z 47.75, A 0, B 90, C 0, E1 0, E2 0, E3 0, E4 0} C_DIS
LIN {X -39.159, Y 234.521, Z 47.75, A 0, B 90, C 0, E1 0, E2 0, E3 0, E4 0} C_DIS
LIN {X -36.946, Y 242.27, Z 47.75, A 0, B 90, C 0, E1 0, E2 0, E3 0, E4 0} C_DIS
LIN {X -34.952, Y 250, Z 50.25, A 0, B 90, C 0, E1 0, E2 0, E3 0, E4 0} C_DIS
LIN {X -32.611, Y 257.69, Z 50.25, A 0, B 90, C 0, E1 0, E2 0, E3 0, E4 0} C_DIS
LIN {X -30.206, Y 265.361, Z 50.25, A 0, B 90, C 0, E1 0, E2 0, E3 0, E4 0} C_DIS
LIN {X -27.741, Y 273.013, Z 50.25, A 0, B 90, C 0, E1 0, E2 0, E3 0, E4 0} C_DIS
LIN {X -25.215, Y 280.645, Z 50.25, A 0, B 90, C 0, E1 0, E2 0, E3 0, E4 0} C_DIS
LIN {X -22.631, Y 288.257, Z 50.25, A 0, B 90, C 0, E1 0, E2 0, E3 0, E4 0} C_DIS
LIN {X -19.99, Y 295.85, Z 50.25, A 0, B 90, C 0, E1 0, E2 0, E3 0, E4 0} C_DIS
LIN {X -17.293, Y 303.422, Z 50.25, A 0, B 90, C 0, E1 0, E2 0, E3 0, E4 0} C_DIS
LIN {X -14.541, Y 310.976, Z 50.25, A 0, B 90, C 0, E1 0, E2 0, E3 0, E4 0} C_DIS
LIN {X -11.736, Y 318.509, Z 50.25, A 0, B 90, C 0, E1 0, E2 0, E3 0, E4 0} C_DIS
LIN {X -8.877, Y 326.023, Z 50.25, A 0, B 90, C 0, E1 0, E2 0, E3 0, E4 0} C_DIS
LIN {X -5.964, Y 333.515, Z 50.25, A 0, B 90, C 0, E1 0, E2 0, E3 0, E4 0} C_DIS
LIN {X -2.997, Y 340.987, Z 50.25, A 0, B 90, C 0, E1 0, E2 0, E3 0, E4 0} C_DIS
LIN {X 0.024, Y 348.437, Z 50.25, A 0, B 90, C 0, E1 0, E2 0, E3 0, E4 0} C_DIS
LIN {X 3.099, Y 355.864, Z 50.25, A 0, B 90, C 0, E1 0, E2 0, E3 0, E4 0} C_DIS
LIN {X 6.229, Y 363.269, Z 50.25, A 0, B 90, C 0, E1 0, E2 0, E3 0, E4 0} C_DIS
LIN {X 10.908, Y 369.563, Z 50.25, A 0, B 90, C 0, E1 0, E2 0, E3 0, E4 0} C_DIS
LIN {X 18.678, Y 369.825, Z 50.25, A 0, B 90, C 0, E1 0, E2 0, E3 0, E4 0} C_DIS
LIN {X 26.067, Y 366.657, Z 50.25, A 0, B 90, C 0, E1 0, E2 0, E3 0, E4 0} C_DIS
LIN {X 33.456, Y 363.49, Z 50.25, A 0, B 90, C 0, E1 0, E2 0, E3 0, E4 0} C_DIS
LIN {X 40.845, Y 360.323, Z 50.25, A 0, B 90, C 0, E1 0, E2 0, E3 0, E4 0} C_DIS
LIN {X 48.234, Y 357.156, Z 50.25, A 0, B 90, C 0, E1 0, E2 0, E3 0, E4 0} C_DIS
LIN {X 55.622, Y 353.989, Z 50.25, A 0, B 90, C 0, E1 0, E2 0, E3 0, E4 0} C_DIS
LIN {X 63.011, Y 350.822, Z 50.25, A 0, B 90, C 0, E1 0, E2 0, E3 0, E4 0} C_DIS
LIN {X 69.478, Y 346.286, Z 50.25, A 0, B 90, C 0, E1 0, E2 0, E3 0, E4 0} C_DIS
LIN {X 69.472, Y 338.66, Z 50.25, A 0, B 90, C 0, E1 0, E2 0, E3 0, E4 0} C_DIS
LIN {X 66.321, Y 331.264, Z 50.25, A 0, B 90, C 0, E1 0, E2 0, E3 0, E4 0} C_DIS
LIN {X 63.23, Y 323.843, Z 50.25, A 0, B 90, C 0, E1 0, E2 0, E3 0, E4 0} C_DIS
LIN {X 60.199, Y 316.398, Z 50.25, A 0, B 90, C 0, E1 0, E2 0, E3 0, E4 0} C_DIS
LIN {X 57.226, Y 308.928, Z 50.25, A 0, B 90, C 0, E1 0, E2 0, E3 0, E4 0} C_DIS
LIN {X 54.313, Y 301.436, Z 50.25, A 0, B 90, C 0, E1 0, E2 0, E3 0, E4 0} C_DIS
LIN {X 51.46, Y 293.921, Z 50.25, A 0, B 90, C 0, E1 0, E2 0, E3 0, E4 0} C_DIS
LIN {X 48.665, Y 286.383, Z 50.25, A 0, B 90, C 0, E1 0, E2 0, E3 0, E4 0} C_DIS
LIN {X 45.928, Y 278.824, Z 50.25, A 0, B 90, C 0, E1 0, E2 0, E3 0, E4 0} C_DIS
LIN {X 43.25, Y 271.245, Z 50.25, A 0, B 90, C 0, E1 0, E2 0, E3 0, E4 0} C_DIS
LIN {X 40.632, Y 263.644, Z 50.25, A 0, B 90, C 0, E1 0, E2 0, E3 0, E4 0} C_DIS
LIN {X 38.075, Y 256.022, Z 50.25, A 0, B 90, C 0, E1 0, E2 0, E3 0, E4 0} C_DIS
LIN {X 35.581, Y 248.38, Z 50.25, A 0, B 90, C 0, E1 0, E2 0, E3 0, E4 0} C_DIS
LIN {X 33.15, Y 240.718, Z 50.25, A 0, B 90, C 0, E1 0, E2 0, E3 0, E4 0} C_DIS
LIN {X 30.785, Y 233.035, Z 50.25, A 0, B 90, C 0, E1 0, E2 0, E3 0, E4 0} C_DIS
LIN {X 28.486, Y 225.331, Z 50.25, A 0, B 90, C 0, E1 0, E2 0, E3 0, E4 0} C_DIS
LIN {X 26.254, Y 217.608, Z 50.25, A 0, B 90, C 0, E1 0, E2 0, E3 0, E4 0} C_DIS
LIN {X 24.092, Y 209.866, Z 50.25, A 0, B 90, C 0, E1 0, E2 0, E3 0, E4 0} C_DIS
LIN {X 22.001, Y 202.104, Z 50.25, A 0, B 90, C 0, E1 0, E2 0, E3 0, E4 0} C_DIS
LIN {X 19.98, Y 194.323, Z 50.25, A 0, B 90, C 0, E1 0, E2 0, E3 0, E4 0} C_DIS
LIN {X 18.033, Y 186.523, Z 50.25, A 0, B 90, C 0, E1 0, E2 0, E3 0, E4 0} C_DIS
LIN {X 16.158, Y 178.706, Z 50.25, A 0, B 90, C 0, E1 0, E2 0, E3 0, E4 0} C_DIS
LIN {X 14.358, Y 170.871, Z 50.25, A 0, B 90, C 0, E1 0, E2 0, E3 0, E4 0} C_DIS
LIN {X 12.633, Y 163.02, Z 50.25, A 0, B 90, C 0, E1 0, E2 0, E3 0, E4 0} C_DIS
LIN {X 10.985, Y 155.151, Z 50.25, A 0, B 90, C 0, E1 0, E2 0, E3 0, E4 0} C_DIS
LIN {X 9.414, Y 147.268, Z 50.25, A 0, B 90, C 0, E1 0, E2 0, E3 0, E4 0} C_DIS
LIN {X 7.92, Y 139.369, Z 50.25, A 0, B 90, C 0, E1 0, E2 0, E3 0, E4 0} C_DIS
LIN {X 6.506, Y 131.455, Z 50.25, A 0, B 90, C 0, E1 0, E2 0, E3 0, E4 0} C_DIS
LIN {X 5.172, Y 123.528, Z 50.25, A 0, B 90, C 0, E1 0, E2 0, E3 0, E4 0} C_DIS
LIN {X 3.917, Y 115.587, Z 50.25, A 0, B 90, C 0, E1 0, E2 0, E3 0, E4 0} C_DIS
LIN {X 2.744, Y 107.634, Z 50.25, A 0, B 90, C 0, E1 0, E2 0, E3 0, E4 0} C_DIS
LIN {X 1.651, Y 99.67, Z 50.25, A 0, B 90, C 0, E1 0, E2 0, E3 0, E4 0} C_DIS
LIN {X 0.64, Y 91.695, Z 50.25, A 0, B 90, C 0, E1 0, E2 0, E3 0, E4 0} C_DIS
LIN {X -0.289, Y 83.71, Z 50.25, A 0, B 90, C 0, E1 0, E2 0, E3 0, E4 0} C_DIS
LIN {X -1.136, Y 75.716, Z 50.25, A 0, B 90, C 0, E1 0, E2 0, E3 0, E4 0} C_DIS
LIN {X -1.899, Y 67.713, Z 50.25, A 0, B 90, C 0, E1 0, E2 0, E3 0, E4 0} C_DIS
LIN {X -2.578, Y 59.703, Z 50.25, A 0, B 90, C 0, E1 0, E2 0, E3 0, E4 0} C_DIS
LIN {X -3.173, Y 51.686, Z 50.25, A 0, B 90, C 0, E1 0, E2 0, E3 0, E4 0} C_DIS
LIN {X -3.684, Y 43.664, Z 50.25, A 0, B 90, C 0, E1 0, E2 0, E3 0, E4 0} C_DIS
LIN {X -4.11, Y 35.636, Z 50.25, A 0, B 90, C 0, E1 0, E2 0, E3 0, E4 0} C_DIS
LIN {X -4.451, Y 27.604, Z 50.25, A 0, B 90, C 0, E1 0, E2 0, E3 0, E4 0} C_DIS
LIN {X -4.706, Y 19.569, Z 50.25, A 0, B 90, C 0, E1 0, E2 0, E3 0, E4 0} C_DIS
LIN {X -4.875, Y 11.532, Z 50.25, A 0, B 90, C 0, E1 0, E2 0, E3 0, E4 0} C_DIS
LIN {X -4.958, Y 3.494, Z 50.25, A 0, B 90, C 0, E1 0, E2 0, E3 0, E4 0} C_DIS
LIN {X -4.953, Y -4.545, Z 50.25, A 0, B 90, C 0, E1 0, E2 0, E3 0, E4 0} C_DIS
LIN {X -4.862, Y -12.584, Z 50.25, A 0, B 90, C 0, E1 0, E2 0, E3 0, E4 0} C_DIS
LIN {X -4.685, Y -20.62, Z 50.25, A 0, B 90, C 0, E1 0, E2 0, E3 0, E4 0} C_DIS
LIN {X -4.421, Y -28.655, Z 50.25, A 0, B 90, C 0, E1 0, E2 0, E3 0, E4 0} C_DIS
LIN {X -4.071, Y -36.686, Z 50.25, A 0, B 90, C 0, E1 0, E2 0, E3 0, E4 0} C_DIS
LIN {X -3.636, Y -44.713, Z 50.25, A 0, B 90, C 0, E1 0, E2 0, E3 0, E4 0} C_DIS
LIN {X -3.115, Y -52.735, Z 50.25, A 0, B 90, C 0, E1 0, E2 0, E3 0, E4 0} C_DIS
LIN {X -2.51, Y -60.752, Z 50.25, A 0, B 90, C 0, E1 0, E2 0, E3 0, E4 0} C_DIS
LIN {X -1.82, Y -68.761, Z 50.25, A 0, B 90, C 0, E1 0, E2 0, E3 0, E4 0} C_DIS
LIN {X -1.045, Y -76.762, Z 50.25, A 0, B 90, C 0, E1 0, E2 0, E3 0, E4 0} C_DIS
LIN {X -0.187, Y -84.755, Z 50.25, A 0, B 90, C 0, E1 0, E2 0, E3 0, E4 0} C_DIS
LIN {X 0.755, Y -92.739, Z 50.25, A 0, B 90, C 0, E1 0, E2 0, E3 0, E4 0} C_DIS
LIN {X 1.779, Y -100.712, Z 50.25, A 0, B 90, C 0, E1 0, E2 0, E3 0, E4 0} C_DIS
LIN {X 2.885, Y -108.675, Z 50.25, A 0, B 90, C 0, E1 0, E2 0, E3 0, E4 0} C_DIS
LIN {X 4.072, Y -116.625, Z 50.25, A 0, B 90, C 0, E1 0, E2 0, E3 0, E4 0} C_DIS
LIN {X 5.34, Y -124.564, Z 50.25, A 0, B 90, C 0, E1 0, E2 0, E3 0, E4 0} C_DIS
LIN {X 6.688, Y -132.489, Z 50.25, A 0, B 90, C 0, E1 0, E2 0, E3 0, E4 0} C_DIS
LIN {X 8.116, Y -140.4, Z 50.25, A 0, B 90, C 0, E1 0, E2 0, E3 0, E4 0} C_DIS
LIN {X 9.622, Y -148.296, Z 50.25, A 0, B 90, C 0, E1 0, E2 0, E3 0, E4 0} C_DIS
LIN {X 11.206, Y -156.178, Z 50.25, A 0, B 90, C 0, E1 0, E2 0, E3 0, E4 0} C_DIS
LIN {X 12.867, Y -164.043, Z 50.25, A 0, B 90, C 0, E1 0, E2 0, E3 0, E4 0} C_DIS
LIN {X 14.603, Y -171.892, Z 50.25, A 0, B 90, C 0, E1 0, E2 0, E3 0, E4 0} C_DIS
LIN {X 16.414, Y -179.725, Z 50.25, A 0, B 90, C 0, E1 0, E2 0, E3 0, E4 0} C_DIS
LIN {X 18.299, Y -187.54, Z 50.25, A 0, B 90, C 0, E1 0, E2 0, E3 0, E4 0} C_DIS
LIN {X 20.255, Y -195.337, Z 50.25, A 0, B 90, C 0, E1 0, E2 0, E3 0, E4 0} C_DIS
LIN {X 22.283, Y -203.116, Z 50.25, A 0, B 90, C 0, E1 0, E2 0, E3 0, E4 0} C_DIS
LIN {X 24.381, Y -210.876, Z 50.25, A 0, B 90, C 0, E1 0, E2 0, E3 0, E4 0} C_DIS
LIN {X 26.549, Y -218.617, Z 50.25, A 0, B 90, C 0, E1 0, E2 0, E3 0, E4 0} C_DIS
LIN {X 28.784, Y -226.339, Z 50.25, A 0, B 90, C 0, E1 0, E2 0, E3 0, E4 0} C_DIS
LIN {X 31.086, Y -234.041, Z 50.25, A 0, B 90, C 0, E1 0, E2 0, E3 0, E4 0} C_DIS
LIN {X 33.454, Y -241.724, Z 50.25, A 0, B 90, C 0, E1 0, E2 0, E3 0, E4 0} C_DIS
LIN {X 35.887, Y -249.385, Z 50.25, A 0, B 90, C 0, E1 0, E2 0, E3 0, E4 0} C_DIS
LIN {X 38.384, Y -257.027, Z 50.25, A 0, B 90, C 0, E1 0, E2 0, E3 0, E4 0} C_DIS
LIN {X 40.944, Y -264.647, Z 50.25, A 0, B 90, C 0, E1 0, E2 0, E3 0, E4 0} C_DIS
LIN {X 43.566, Y -272.247, Z 50.25, A 0, B 90, C 0, E1 0, E2 0, E3 0, E4 0} C_DIS
LIN {X 46.249, Y -279.825, Z 50.25, A 0, B 90, C 0, E1 0, E2 0, E3 0, E4 0} C_DIS
LIN {X 48.992, Y -287.381, Z 50.25, A 0, B 90, C 0, E1 0, E2 0, E3 0, E4 0} C_DIS
LIN {X 51.795, Y -294.916, Z 50.25, A 0, B 90, C 0, E1 0, E2 0, E3 0, E4 0} C_DIS
LIN {X 54.658, Y -302.427, Z 50.25, A 0, B 90, C 0, E1 0, E2 0, E3 0, E4 0} C_DIS
LIN {X 57.581, Y -309.916, Z 50.25, A 0, B 90, C 0, E1 0, E2 0, E3 0, E4 0} C_DIS
LIN {X 60.565, Y -317.38, Z 50.25, A 0, B 90, C 0, E1 0, E2 0, E3 0, E4 0} C_DIS
LIN {X 63.609, Y -324.821, Z 50.25, A 0, B 90, C 0, E1 0, E2 0, E3 0, E4 0} C_DIS
LIN {X 66.714, Y -332.236, Z 50.25, A 0, B 90, C 0, E1 0, E2 0, E3 0, E4 0} C_DIS
LIN {X 69.88, Y -339.625, Z 50.25, A 0, B 90, C 0, E1 0, E2 0, E3 0, E4 0} C_DIS
LIN {X 68.854, Y -347.134, Z 50.25, A 0, B 90, C 0, E1 0, E2 0, E3 0, E4 0} C_DIS
LIN {X 62.044, Y -351.24, Z 50.25, A 0, B 90, C 0, E1 0, E2 0, E3 0, E4 0} C_DIS
LIN {X 54.656, Y -354.407, Z 50.25, A 0, B 90, C 0, E1 0, E2 0, E3 0, E4 0} C_DIS
LIN {X 47.267, Y -357.574, Z 50.25, A 0, B 90, C 0, E1 0, E2 0, E3 0, E4 0} C_DIS
LIN {X 39.878, Y -360.741, Z 50.25, A 0, B 90, C 0, E1 0, E2 0, E3 0, E4 0} C_DIS
LIN {X 32.489, Y -363.908, Z 50.25, A 0, B 90, C 0, E1 0, E2 0, E3 0, E4 0} C_DIS
LIN {X 25.1, Y -367.075, Z 50.25, A 0, B 90, C 0, E1 0, E2 0, E3 0, E4 0} C_DIS
LIN {X 17.688, Y -370.151, Z 50.25, A 0, B 90, C 0, E1 0, E2 0, E3 0, E4 0} C_DIS
LIN {X 10.017, Y -369.007, Z 50.25, A 0, B 90, C 0, E1 0, E2 0, E3 0, E4 0} C_DIS
LIN {X 5.816, Y -362.304, Z 50.25, A 0, B 90, C 0, E1 0, E2 0, E3 0, E4 0} C_DIS
LIN {X 2.693, Y -354.897, Z 50.25, A 0, B 90, C 0, E1 0, E2 0, E3 0, E4 0} C_DIS
LIN {X -0.375, Y -347.466, Z 50.25, A 0, B 90, C 0, E1 0, E2 0, E3 0, E4 0} C_DIS
LIN {X -3.389, Y -340.014, Z 50.25, A 0, B 90, C 0, E1 0, E2 0, E3 0, E4 0} C_DIS
LIN {X -6.349, Y -332.54, Z 50.25, A 0, B 90, C 0, E1 0, E2 0, E3 0, E4 0} C_DIS
LIN {X -9.255, Y -325.044, Z 50.25, A 0, B 90, C 0, E1 0, E2 0, E3 0, E4 0} C_DIS
LIN {X -12.107, Y -317.528, Z 50.25, A 0, B 90, C 0, E1 0, E2 0, E3 0, E4 0} C_DIS
LIN {X -14.905, Y -309.992, Z 50.25, A 0, B 90, C 0, E1 0, E2 0, E3 0, E4 0} C_DIS
LIN {X -17.649, Y -302.436, Z 50.25, A 0, B 90, C 0, E1 0, E2 0, E3 0, E4 0} C_DIS
LIN {X -20.339, Y -294.86, Z 50.25, A 0, B 90, C 0, E1 0, E2 0, E3 0, E4 0} C_DIS
LIN {X -22.972, Y -287.265, Z 50.25, A 0, B 90, C 0, E1 0, E2 0, E3 0, E4 0} C_DIS
LIN {X -25.548, Y -279.65, Z 50.25, A 0, B 90, C 0, E1 0, E2 0, E3 0, E4 0} C_DIS
LIN {X -28.065, Y -272.015, Z 50.25, A 0, B 90, C 0, E1 0, E2 0, E3 0, E4 0} C_DIS
LIN {X -30.522, Y -264.361, Z 50.25, A 0, B 90, C 0, E1 0, E2 0, E3 0, E4 0} C_DIS
LIN {X -32.918, Y -256.687, Z 50.25, A 0, B 90, C 0, E1 0, E2 0, E3 0, E4 0} C_DIS
LIN {X -35.252, Y -248.995, Z 50.25, A 0, B 90, C 0, E1 0, E2 0, E3 0, E4 0} C_DIS
LIN {X -37.522, Y -241.283, Z 50.25, A 0, B 90, C 0, E1 0, E2 0, E3 0, E4 0} C_DIS
LIN {X -39.728, Y -233.553, Z 50.25, A 0, B 90, C 0, E1 0, E2 0, E3 0, E4 0} C_DIS
LIN {X -41.87, Y -225.804, Z 50.25, A 0, B 90, C 0, E1 0, E2 0, E3 0, E4 0} C_DIS
LIN {X -43.945, Y -218.038, Z 50.25, A 0, B 90, C 0, E1 0, E2 0, E3 0, E4 0} C_DIS
LIN {X -45.954, Y -210.254, Z 50.25, A 0, B 90, C 0, E1 0, E2 0, E3 0, E4 0} C_DIS
LIN {X -47.896, Y -202.453, Z 50.25, A 0, B 90, C 0, E1 0, E2 0, E3 0, E4 0} C_DIS
LIN {X -49.77, Y -194.635, Z 50.25, A 0, B 90, C 0, E1 0, E2 0, E3 0, E4 0} C_DIS
LIN {X -51.575, Y -186.802, Z 50.25, A 0, B 90, C 0, E1 0, E2 0, E3 0, E4 0} C_DIS
LIN {X -53.311, Y -178.953, Z 50.25, A 0, B 90, C 0, E1 0, E2 0, E3 0, E4 0} C_DIS
LIN {X -54.977, Y -171.088, Z 50.25, A 0, B 90, C 0, E1 0, E2 0, E3 0, E4 0} C_DIS
LIN {X -56.572, Y -163.209, Z 50.25, A 0, B 90, C 0, E1 0, E2 0, E3 0, E4 0} C_DIS
LIN {X -58.095, Y -155.316, Z 50.25, A 0, B 90, C 0, E1 0, E2 0, E3 0, E4 0} C_DIS
LIN {X -59.547, Y -147.409, Z 50.25, A 0, B 90, C 0, E1 0, E2 0, E3 0, E4 0} C_DIS
LIN {X -60.925, Y -139.489, Z 50.25, A 0, B 90, C 0, E1 0, E2 0, E3 0, E4 0} C_DIS
LIN {X -62.23, Y -131.557, Z 50.25, A 0, B 90, C 0, E1 0, E2 0, E3 0, E4 0} C_DIS
LIN {X -63.462, Y -123.613, Z 50.25, A 0, B 90, C 0, E1 0, E2 0, E3 0, E4 0} C_DIS
LIN {X -64.619, Y -115.658, Z 50.25, A 0, B 90, C 0, E1 0, E2 0, E3 0, E4 0} C_DIS
LIN {X -65.7, Y -107.692, Z 50.25, A 0, B 90, C 0, E1 0, E2 0, E3 0, E4 0} C_DIS
LIN {X -66.707, Y -99.716, Z 50.25, A 0, B 90, C 0, E1 0, E2 0, E3 0, E4 0} C_DIS
LIN {X -67.637, Y -91.731, Z 50.25, A 0, B 90, C 0, E1 0, E2 0, E3 0, E4 0} C_DIS
LIN {X -68.492, Y -83.738, Z 50.25, A 0, B 90, C 0, E1 0, E2 0, E3 0, E4 0} C_DIS
LIN {X -69.27, Y -75.737, Z 50.25, A 0, B 90, C 0, E1 0, E2 0, E3 0, E4 0} C_DIS
LIN {X -69.972, Y -67.729, Z 50.25, A 0, B 90, C 0, E1 0, E2 0, E3 0, E4 0} C_DIS
LIN {X -70.597, Y -59.714, Z 50.25, A 0, B 90, C 0, E1 0, E2 0, E3 0, E4 0} C_DIS
LIN {X -71.144, Y -51.694, Z 50.25, A 0, B 90, C 0, E1 0, E2 0, E3 0, E4 0} C_DIS
LIN {X -71.613, Y -43.669, Z 50.25, A 0, B 90, C 0, E1 0, E2 0, E3 0, E4 0} C_DIS
LIN {X -72.004, Y -35.639, Z 50.25, A 0, B 90, C 0, E1 0, E2 0, E3 0, E4 0} C_DIS
LIN {X -72.317, Y -27.606, Z 50.25, A 0, B 90, C 0, E1 0, E2 0, E3 0, E4 0} C_DIS
LIN {X -72.551, Y -19.571, Z 50.25, A 0, B 90, C 0, E1 0, E2 0, E3 0, E4 0} C_DIS
LIN {X -72.705, Y -11.533, Z 50.25, A 0, B 90, C 0, E1 0, E2 0, E3 0, E4 0} C_DIS
LIN {X -72.78, Y -3.495, Z 50.25, A 0, B 90, C 0, E1 0, E2 0, E3 0, E4 0} C_DIS
LIN {X -72.775, Y 4.544, Z 50.25, A 0, B 90, C 0, E1 0, E2 0, E3 0, E4 0} C_DIS
LIN {X -72.691, Y 12.583, Z 50.25, A 0, B 90, C 0, E1 0, E2 0, E3 0, E4 0} C_DIS
LIN {X -72.527, Y 20.62, Z 50.25, A 0, B 90, C 0, E1 0, E2 0, E3 0, E4 0} C_DIS
LIN {X -72.283, Y 28.655, Z 50.25, A 0, B 90, C 0, E1 0, E2 0, E3 0, E4 0} C_DIS
LIN {X -71.961, Y 36.687, Z 50.25, A 0, B 90, C 0, E1 0, E2 0, E3 0, E4 0} C_DIS
LIN {X -71.56, Y 44.716, Z 50.25, A 0, B 90, C 0, E1 0, E2 0, E3 0, E4 0} C_DIS
LIN {X -71.081, Y 52.741, Z 50.25, A 0, B 90, C 0, E1 0, E2 0, E3 0, E4 0} C_DIS
LIN {X -70.524, Y 60.761, Z 50.25, A 0, B 90, C 0, E1 0, E2 0, E3 0, E4 0} C_DIS
LIN {X -69.89, Y 68.774, Z 50.25, A 0, B 90, C 0, E1 0, E2 0, E3 0, E4 0} C_DIS
LIN {X -69.178, Y 76.782, Z 50.25, A 0, B 90, C 0, E1 0, E2 0, E3 0, E4 0} C_DIS
LIN {X -68.389, Y 84.782, Z 50.25, A 0, B 90, C 0, E1 0, E2 0, E3 0, E4 0} C_DIS
LIN {X -67.524, Y 92.774, Z 50.25, A 0, B 90, C 0, E1 0, E2 0, E3 0, E4 0} C_DIS
LIN {X -66.583, Y 100.758, Z 50.25, A 0, B 90, C 0, E1 0, E2 0, E3 0, E4 0} C_DIS
LIN {X -65.565, Y 108.732, Z 50.25, A 0, B 90, C 0, E1 0, E2 0, E3 0, E4 0} C_DIS
LIN {X -64.473, Y 116.696, Z 50.25, A 0, B 90, C 0, E1 0, E2 0, E3 0, E4 0} C_DIS
LIN {X -63.305, Y 124.65, Z 50.25, A 0, B 90, C 0, E1 0, E2 0, E3 0, E4 0} C_DIS
LIN {X -62.063, Y 132.592, Z 50.25, A 0, B 90, C 0, E1 0, E2 0, E3 0, E4 0} C_DIS
LIN {X -60.747, Y 140.523, Z 50.25, A 0, B 90, C 0, E1 0, E2 0, E3 0, E4 0} C_DIS
LIN {X -59.358, Y 148.441, Z 50.25, A 0, B 90, C 0, E1 0, E2 0, E3 0, E4 0} C_DIS
LIN {X -57.897, Y 156.346, Z 50.25, A 0, B 90, C 0, E1 0, E2 0, E3 0, E4 0} C_DIS
LIN {X -56.363, Y 164.237, Z 50.25, A 0, B 90, C 0, E1 0, E2 0, E3 0, E4 0} C_DIS
LIN {X -54.759, Y 172.114, Z 50.25, A 0, B 90, C 0, E1 0, E2 0, E3 0, E4 0} C_DIS
LIN {X -53.084, Y 179.977, Z 50.25, A 0, B 90, C 0, E1 0, E2 0, E3 0, E4 0} C_DIS
LIN {X -51.339, Y 187.824, Z 50.25, A 0, B 90, C 0, E1 0, E2 0, E3 0, E4 0} C_DIS
LIN {X -49.526, Y 195.656, Z 50.25, A 0, B 90, C 0, E1 0, E2 0, E3 0, E4 0} C_DIS
LIN {X -47.644, Y 203.471, Z 50.25, A 0, B 90, C 0, E1 0, E2 0, E3 0, E4 0} C_DIS
LIN {X -45.694, Y 211.27, Z 50.25, A 0, B 90, C 0, E1 0, E2 0, E3 0, E4 0} C_DIS
LIN {X -43.677, Y 219.052, Z 50.25, A 0, B 90, C 0, E1 0, E2 0, E3 0, E4 0} C_DIS
LIN {X -41.594, Y 226.816, Z 50.25, A 0, B 90, C 0, E1 0, E2 0, E3 0, E4 0} C_DIS
LIN {X -39.445, Y 234.563, Z 50.25, A 0, B 90, C 0, E1 0, E2 0, E3 0, E4 0} C_DIS
LIN {X -37.231, Y 242.291, Z 50.25, A 0, B 90, C 0, E1 0, E2 0, E3 0, E4 0} C_DIS
LIN {X -35.236, Y 250, Z 52.75, A 0, B 90, C 0, E1 0, E2 0, E3 0, E4 0} C_DIS
LIN {X -32.894, Y 257.669, Z 52.75, A 0, B 90, C 0, E1 0, E2 0, E3 0, E4 0} C_DIS
LIN {X -30.489, Y 265.319, Z 52.75, A 0, B 90, C 0, E1 0, E2 0, E3 0, E4 0} C_DIS
LIN {X -28.023, Y 272.949, Z 52.75, A 0, B 90, C 0, E1 0, E2 0, E3 0, E4 0} C_DIS
LIN {X -25.498, Y 280.56, Z 52.75, A 0, B 90, C 0, E1 0, E2 0, E3 0, E4 0} C_DIS
LIN {X -22.914, Y 288.152, Z 52.75, A 0, B 90, C 0, E1 0, E2 0, E3 0, E4 0} C_DIS
LIN {X -20.273, Y 295.723, Z 52.75, A 0, B 90, C 0, E1 0, E2 0, E3 0, E4 0} C_DIS
LIN {X -17.577, Y 303.275, Z 52.75, A 0, B 90, C 0, E1 0, E2 0, E3 0, E4 0} C_DIS
LIN {X -14.826, Y 310.808, Z 52.75, A 0, B 90, C 0, E1 0, E2 0, E3 0, E4 0} C_DIS
LIN {X -12.022, Y 318.321, Z 52.75, A 0, B 90, C 0, E1 0, E2 0, E3 0, E4 0} C_DIS
LIN {X -9.165, Y 325.813, Z 52.75, A 0, B 90, C 0, E1 0, E2 0, E3 0, E4 0} C_DIS
LIN {X -6.254, Y 333.285, Z 52.75, A 0, B 90, C 0, E1 0, E2 0, E3 0, E4 0} C_DIS
LIN {X -3.289, Y 340.736, Z 52.75, A 0, B 90, C 0, E1 0, E2 0, E3 0, E4 0} C_DIS
LIN {X -0.27, Y 348.165, Z 52.75, A 0, B 90, C 0, E1 0, E2 0, E3 0, E4 0} C_DIS
LIN {X 2.803, Y 355.571, Z 52.75, A 0, B 90, C 0, E1 0, E2 0, E3 0, E4 0} C_DIS
LIN {X 5.932, Y 362.955, Z 52.75, A 0, B 90, C 0, E1 0, E2 0, E3 0, E4 0} C_DIS
LIN {X 10.705, Y 369.137, Z 52.75, A 0, B 90, C 0, E1 0, E2 0, E3 0, E4 0} C_DIS
LIN {X 18.466, Y 369.242, Z 52.75, A 0, B 90, C 0, E1 0, E2 0, E3 0, E4 0} C_DIS
LIN {X 25.836, Y 366.081, Z 52.75, A 0, B 90, C 0, E1 0, E2 0, E3 0, E4 0} C_DIS
LIN {X 33.205, Y 362.92, Z 52.75, A 0, B 90, C 0, E1 0, E2 0, E3 0, E4 0} C_DIS
LIN {X 40.575, Y 359.759, Z 52.75, A 0, B 90, C 0, E1 0, E2 0, E3 0, E4 0} C_DIS
LIN {X 47.945, Y 356.598, Z 52.75, A 0, B 90, C 0, E1 0, E2 0, E3 0, E4 0} C_DIS
LIN {X 55.314, Y 353.437, Z 52.75, A 0, B 90, C 0, E1 0, E2 0, E3 0, E4 0} C_DIS
LIN {X 62.684, Y 350.276, Z 52.75, A 0, B 90, C 0, E1 0, E2 0, E3 0, E4 0} C_DIS
LIN {X 68.308, Y 344.885, Z 52.75, A 0, B 90, C 0, E1 0, E2 0, E3 0, E4 0} C_DIS
LIN {X 66.887, Y 337.241, Z 52.75, A 0, B 90, C 0, E1 0, E2 0, E3 0, E4 0} C_DIS
LIN {X 63.752, Y 329.86, Z 52.75, A 0, B 90, C 0, E1 0, E2 0, E3 0, E4 0} C_DIS
LIN {X 60.676, Y 322.454, Z 52.75, A 0, B 90, C 0, E1 0, E2 0, E3 0, E4 0} C_DIS
LIN {X 57.66, Y 315.024, Z 52.75, A 0, B 90, C 0, E1 0, E2 0, E3 0, E4 0} C_DIS
LIN {X 54.702, Y 307.571, Z 52.75, A 0, B 90, C 0, E1 0, E2 0, E3 0, E4 0} C_DIS
LIN {X 51.804, Y 300.094, Z 52.75, A 0, B 90, C 0, E1 0, E2 0, E3 0, E4 0} C_DIS
LIN {X 48.965, Y 292.594, Z 52.75, A 0, B 90, C 0, E1 0, E2 0, E3 0, E4 0} C_DIS
LIN {X 46.184, Y 285.073, Z 52.75, A 0, B 90, C 0, E1 0, E2 0, E3 0, E4 0} C_DIS
LIN {X 43.461, Y 277.53, Z 52.75, A 0, B 90, C 0, E1 0, E2 0, E3 0, E4 0} C_DIS
LIN {X 40.797, Y 269.967, Z 52.75, A 0, B 90, C 0, E1 0, E2 0, E3 0, E4 0} C_DIS
LIN {X 38.193, Y 262.383, Z 52.75, A 0, B 90, C 0, E1 0, E2 0, E3 0, E4 0} C_DIS
LIN {X 35.65, Y 254.778, Z 52.75, A 0, B 90, C 0, E1 0, E2 0, E3 0, E4 0} C_DIS
LIN {X 33.169, Y 247.152, Z 52.75, A 0, B 90, C 0, E1 0, E2 0, E3 0, E4 0} C_DIS
LIN {X 30.752, Y 239.506, Z 52.75, A 0, B 90, C 0, E1 0, E2 0, E3 0, E4 0} C_DIS
LIN {X 28.4, Y 231.84, Z 52.75, A 0, B 90, C 0, E1 0, E2 0, E3 0, E4 0} C_DIS
LIN {X 26.114, Y 224.153, Z 52.75, A 0, B 90, C 0, E1 0, E2 0, E3 0, E4 0} C_DIS
LIN {X 23.897, Y 216.447, Z 52.75, A 0, B 90, C 0, E1 0, E2 0, E3 0, E4 0} C_DIS
LIN {X 21.748, Y 208.722, Z 52.75, A 0, B 90, C 0, E1 0, E2 0, E3 0, E4 0} C_DIS
LIN {X 19.67, Y 200.977, Z 52.75, A 0, B 90, C 0, E1 0, E2 0, E3 0, E4 0} C_DIS
LIN {X 17.662, Y 193.213, Z 52.75, A 0, B 90, C 0, E1 0, E2 0, E3 0, E4 0} C_DIS
LIN {X 15.728, Y 185.431, Z 52.75, A 0, B 90, C 0, E1 0, E2 0, E3 0, E4 0} C_DIS
LIN {X 13.866, Y 177.631, Z 52.75, A 0, B 90, C 0, E1 0, E2 0, E3 0, E4 0} C_DIS
LIN {X 12.079, Y 169.814, Z 52.75, A 0, B 90, C 0, E1 0, E2 0, E3 0, E4 0} C_DIS
LIN {X 10.366, Y 161.98, Z 52.75, A 0, B 90, C 0, E1 0, E2 0, E3 0, E4 0} C_DIS
LIN {X 8.73, Y 154.13, Z 52.75, A 0, B 90, C 0, E1 0, E2 0, E3 0, E4 0} C_DIS
LIN {X 7.171, Y 146.264, Z 52.75, A 0, B 90, C 0, E1 0, E2 0, E3 0, E4 0} C_DIS
LIN {X 5.69, Y 138.383, Z 52.75, A 0, B 90, C 0, E1 0, E2 0, E3 0, E4 0} C_DIS
LIN {X 4.287, Y 130.487, Z 52.75, A 0, B 90, C 0, E1 0, E2 0, E3 0, E4 0} C_DIS
LIN {X 2.965, Y 122.578, Z 52.75, A 0, B 90, C 0, E1 0, E2 0, E3 0, E4 0} C_DIS
LIN {X 1.721, Y 114.656, Z 52.75, A 0, B 90, C 0, E1 0, E2 0, E3 0, E4 0} C_DIS
LIN {X 0.559, Y 106.722, Z 52.75, A 0, B 90, C 0, E1 0, E2 0, E3 0, E4 0} C_DIS
LIN {X -0.523, Y 98.777, Z 52.75, A 0, B 90, C 0, E1 0, E2 0, E3 0, E4 0} C_DIS
LIN {X -1.524, Y 90.82, Z 52.75, A 0, B 90, C 0, E1 0, E2 0, E3 0, E4 0} C_DIS
LIN {X -2.442, Y 82.854, Z 52.75, A 0, B 90, C 0, E1 0, E2 0, E3 0, E4 0} C_DIS
LIN {X -3.279, Y 74.879, Z 52.75, A 0, B 90, C 0, E1 0, E2 0, E3 0, E4 0} C_DIS
LIN {X -4.032, Y 66.895, Z 52.75, A 0, B 90, C 0, E1 0, E2 0, E3 0, E4 0} C_DIS
LIN {X -4.702, Y 58.904, Z 52.75, A 0, B 90, C 0, E1 0, E2 0, E3 0, E4 0} C_DIS
LIN {X -5.288, Y 50.907, Z 52.75, A 0, B 90, C 0, E1 0, E2 0, E3 0, E4 0} C_DIS
LIN {X -5.79, Y 42.904, Z 52.75, A 0, B 90, C 0, E1 0, E2 0, E3 0, E4 0} C_DIS
LIN {X -6.207, Y 34.896, Z 52.75, A 0, B 90, C 0, E1 0, E2 0, E3 0, E4 0} C_DIS
LIN {X -6.54, Y 26.884, Z 52.75, A 0, B 90, C 0, E1 0, E2 0, E3 0, E4 0} C_DIS
LIN {X -6.787, Y 18.869, Z 52.75, A 0, B 90, C 0, E1 0, E2 0, E3 0, E4 0} C_DIS
LIN {X -6.948, Y 10.851, Z 52.75, A 0, B 90, C 0, E1 0, E2 0, E3 0, E4 0} C_DIS
LIN {X -7.024, Y 2.833, Z 52.75, A 0, B 90, C 0, E1 0, E2 0, E3 0, E4 0} C_DIS
LIN {X -7.012, Y -5.186, Z 52.75, A 0, B 90, C 0, E1 0, E2 0, E3 0, E4 0} C_DIS
LIN {X -6.915, Y -13.205, Z 52.75, A 0, B 90, C 0, E1 0, E2 0, E3 0, E4 0} C_DIS
LIN {X -6.731, Y -21.221, Z 52.75, A 0, B 90, C 0, E1 0, E2 0, E3 0, E4 0} C_DIS
LIN {X -6.462, Y -29.236, Z 52.75, A 0, B 90, C 0, E1 0, E2 0, E3 0, E4 0} C_DIS
LIN {X -6.106, Y -37.247, Z 52.75, A 0, B 90, C 0, E1 0, E2 0, E3 0, E4 0} C_DIS
LIN {X -5.666, Y -45.254, Z 52.75, A 0, B 90, C 0, E1 0, E2 0, E3 0, E4 0} C_DIS
LIN {X -5.141, Y -53.255, Z 52.75, A 0, B 90, C 0, E1 0, E2 0, E3 0, E4 0} C_DIS
LIN {X -4.531, Y -61.251, Z 52.75, A 0, B 90, C 0, E1 0, E2 0, E3 0, E4 0} C_DIS
LIN {X -3.837, Y -69.24, Z 52.75, A 0, B 90, C 0, E1 0, E2 0, E3 0, E4 0} C_DIS
LIN {X -3.058, Y -77.221, Z 52.75, A 0, B 90, C 0, E1 0, E2 0, E3 0, E4 0} C_DIS
LIN {X -2.196, Y -85.194, Z 52.75, A 0, B 90, C 0, E1 0, E2 0, E3 0, E4 0} C_DIS
LIN {X -1.252, Y -93.157, Z 52.75, A 0, B 90, C 0, E1 0, E2 0, E3 0, E4 0} C_DIS
LIN {X -0.225, Y -101.11, Z 52.75, A 0, B 90, C 0, E1 0, E2 0, E3 0, E4 0} C_DIS
LIN {X 0.884, Y -109.052, Z 52.75, A 0, B 90, C 0, E1 0, E2 0, E3 0, E4 0} C_DIS
LIN {X 2.073, Y -116.982, Z 52.75, A 0, B 90, C 0, E1 0, E2 0, E3 0, E4 0} C_DIS
LIN {X 3.343, Y -124.9, Z 52.75, A 0, B 90, C 0, E1 0, E2 0, E3 0, E4 0} C_DIS
LIN {X 4.692, Y -132.804, Z 52.75, A 0, B 90, C 0, E1 0, E2 0, E3 0, E4 0} C_DIS
LIN {X 6.121, Y -140.695, Z 52.75, A 0, B 90, C 0, E1 0, E2 0, E3 0, E4 0} C_DIS
LIN {X 7.628, Y -148.571, Z 52.75, A 0, B 90, C 0, E1 0, E2 0, E3 0, E4 0} C_DIS
LIN {X 9.213, Y -156.432, Z 52.75, A 0, B 90, C 0, E1 0, E2 0, E3 0, E4 0} C_DIS
LIN {X 10.874, Y -164.277, Z 52.75, A 0, B 90, C 0, E1 0, E2 0, E3 0, E4 0} C_DIS
LIN {X 12.61, Y -172.105, Z 52.75, A 0, B 90, C 0, E1 0, E2 0, E3 0, E4 0} C_DIS
LIN {X 14.421, Y -179.917, Z 52.75, A 0, B 90, C 0, E1 0, E2 0, E3 0, E4 0} C_DIS
LIN {X 16.304, Y -187.712, Z 52.75, A 0, B 90, C 0, E1 0, E2 0, E3 0, E4 0} C_DIS
LIN {X 18.26, Y -195.489, Z 52.75, A 0, B 90, C 0, E1 0, E2 0, E3 0, E4 0} C_DIS
LIN {X 20.286, Y -203.247, Z 52.75, A 0, B 90, C 0, E1 0, E2 0, E3 0, E4 0} C_DIS
LIN {X 22.382, Y -210.987, Z 52.75, A 0, B 90, C 0, E1 0, E2 0, E3 0, E4 0} C_DIS
LIN {X 24.547, Y -218.709, Z 52.75, A 0, B 90, C 0, E1 0, E2 0, E3 0, E4 0} C_DIS
LIN {X 26.78, Y -226.411, Z 52.75, A 0, B 90, C 0, E1 0, E2 0, E3 0, E4 0} C_DIS
LIN {X 29.079, Y -234.093, Z 52.75, A 0, B 90, C 0, E1 0, E2 0, E3 0, E4 0} C_DIS
LIN {X 31.444, Y -241.755, Z 52.75, A 0, B 90, C 0, E1 0, E2 0, E3 0, E4 0} C_DIS
LIN {X 33.873, Y -249.397, Z 52.75, A 0, B 90, C 0, E1 0, E2 0, E3 0, E4 0} C_DIS
LIN {X 36.367, Y -257.019, Z 52.75, A 0, B 90, C 0, E1 0, E2 0, E3 0, E4 0} C_DIS
LIN {X 38.922, Y -264.619, Z 52.75, A 0, B 90, C 0, E1 0, E2 0, E3 0, E4 0} C_DIS
LIN {X 41.54, Y -272.199, Z 52.75, A 0, B 90, C 0, E1 0, E2 0, E3 0, E4 0} C_DIS
LIN {X 44.218, Y -279.758, Z 52.75, A 0, B 90, C 0, E1 0, E2 0, E3 0, E4 0} C_DIS
LIN {X 46.957, Y -287.294, Z 52.75, A 0, B 90, C 0, E1 0, E2 0, E3 0, E4 0} C_DIS
LIN {X 49.755, Y -294.809, Z 52.75, A 0, B 90, C 0, E1 0, E2 0, E3 0, E4 0} C_DIS
LIN {X 52.613, Y -302.302, Z 52.75, A 0, B 90, C 0, E1 0, E2 0, E3 0, E4 0} C_DIS
LIN {X 55.532, Y -309.771, Z 52.75, A 0, B 90, C 0, E1 0, E2 0, E3 0, E4 0} C_DIS
LIN {X 58.511, Y -317.216, Z 52.75, A 0, B 90, C 0, E1 0, E2 0, E3 0, E4 0} C_DIS
LIN {X 61.549, Y -324.637, Z 52.75, A 0, B 90, C 0, E1 0, E2 0, E3 0, E4 0} C_DIS
LIN {X 64.649, Y -332.032, Z 52.75, A 0, B 90, C 0, E1 0, E2 0, E3 0, E4 0} C_DIS
LIN {X 67.808, Y -339.403, Z 52.75, A 0, B 90, C 0, E1 0, E2 0, E3 0, E4 0} C_DIS
LIN {X 67.189, Y -346.947, Z 52.75, A 0, B 90, C 0, E1 0, E2 0, E3 0, E4 0} C_DIS
LIN {X 60.52, Y -351.207, Z 52.75, A 0, B 90, C 0, E1 0, E2 0, E3 0, E4 0} C_DIS
LIN {X 53.15, Y -354.368, Z 52.75, A 0, B 90, C 0, E1 0, E2 0, E3 0, E4 0} C_DIS
LIN {X 45.781, Y -357.529, Z 52.75, A 0, B 90, C 0, E1 0, E2 0, E3 0, E4 0} C_DIS
LIN {X 38.411, Y -360.69, Z 52.75, A 0, B 90, C 0, E1 0, E2 0, E3 0, E4 0} C_DIS
LIN {X 31.041, Y -363.851, Z 52.75, A 0, B 90, C 0, E1 0, E2 0, E3 0, E4 0} C_DIS
LIN {X 23.672, Y -367.012, Z 52.75, A 0, B 90, C 0, E1 0, E2 0, E3 0, E4 0} C_DIS
LIN {X 16.209, Y -369.851, Z 52.75, A 0, B 90, C 0, E1 0, E2 0, E3 0, E4 0} C_DIS
LIN {X 8.786, Y -367.789, Z 52.75, A 0, B 90, C 0, E1 0, E2 0, E3 0, E4 0} C_DIS
LIN {X 5.008, Y -360.792, Z 52.75, A 0, B 90, C 0, E1 0, E2 0, E3 0, E4 0} C_DIS
LIN {X 1.895, Y -353.402, Z 52.75, A 0, B 90, C 0, E1 0, E2 0, E3 0, E4 0} C_DIS
LIN {X -1.163, Y -345.989, Z 52.75, A 0, B 90, C 0, E1 0, E2 0, E3 0, E4 0} C_DIS
LIN {X -4.166, Y -338.554, Z 52.75, A 0, B 90, C 0, E1 0, E2 0, E3 0, E4 0} C_DIS
LIN {X -7.115, Y -331.097, Z 52.75, A 0, B 90, C 0, E1 0, E2 0, E3 0, E4 0} C_DIS
LIN {X -10.011, Y -323.619, Z 52.75, A 0, B 90, C 0, E1 0, E2 0, E3 0, E4 0} C_DIS
LIN {X -12.852, Y -316.12, Z 52.75, A 0, B 90, C 0, E1 0, E2 0, E3 0, E4 0} C_DIS
LIN {X -15.64, Y -308.602, Z 52.75, A 0, B 90, C 0, E1 0, E2 0, E3 0, E4 0} C_DIS
LIN {X -18.375, Y -301.063, Z 52.75, A 0, B 90, C 0, E1 0, E2 0, E3 0, E4 0} C_DIS
LIN {X -21.054, Y -293.505, Z 52.75, A 0, B 90, C 0, E1 0, E2 0, E3 0, E4 0} C_DIS
LIN {X -23.678, Y -285.928, Z 52.75, A 0, B 90, C 0, E1 0, E2 0, E3 0, E4 0} C_DIS
LIN {X -26.244, Y -278.33, Z 52.75, A 0, B 90, C 0, E1 0, E2 0, E3 0, E4 0} C_DIS
LIN {X -28.752, Y -270.714, Z 52.75, A 0, B 90, C 0, E1 0, E2 0, E3 0, E4 0} C_DIS
LIN {X -31.199, Y -263.077, Z 52.75, A 0, B 90, C 0, E1 0, E2 0, E3 0, E4 0} C_DIS
LIN {X -33.586, Y -255.422, Z 52.75, A 0, B 90, C 0, E1 0, E2 0, E3 0, E4 0} C_DIS
LIN {X -35.91, Y -247.747, Z 52.75, A 0, B 90, C 0, E1 0, E2 0, E3 0, E4 0} C_DIS
LIN {X -38.17, Y -240.053, Z 52.75, A 0, B 90, C 0, E1 0, E2 0, E3 0, E4 0} C_DIS
LIN {X -40.367, Y -232.341, Z 52.75, A 0, B 90, C 0, E1 0, E2 0, E3 0, E4 0} C_DIS
LIN {X -42.499, Y -224.611, Z 52.75, A 0, B 90, C 0, E1 0, E2 0, E3 0, E4 0} C_DIS
LIN {X -44.565, Y -216.862, Z 52.75, A 0, B 90, C 0, E1 0, E2 0, E3 0, E4 0} C_DIS
LIN {X -46.564, Y -209.097, Z 52.75, A 0, B 90, C 0, E1 0, E2 0, E3 0, E4 0} C_DIS
LIN {X -48.497, Y -201.314, Z 52.75, A 0, B 90, C 0, E1 0, E2 0, E3 0, E4 0} C_DIS
LIN {X -50.361, Y -193.515, Z 52.75, A 0, B 90, C 0, E1 0, E2 0, E3 0, E4 0} C_DIS
LIN {X -52.157, Y -185.7, Z 52.75, A 0, B 90, C 0, E1 0, E2 0, E3 0, E4 0} C_DIS
LIN {X -53.884, Y -177.869, Z 52.75, A 0, B 90, C 0, E1 0, E2 0, E3 0, E4 0} C_DIS
LIN {X -55.541, Y -170.023, Z 52.75, A 0, B 90, C 0, E1 0, E2 0, E3 0, E4 0} C_DIS
LIN {X -57.127, Y -162.162, Z 52.75, A 0, B 90, C 0, E1 0, E2 0, E3 0, E4 0} C_DIS
LIN {X -58.642, Y -154.288, Z 52.75, A 0, B 90, C 0, E1 0, E2 0, E3 0, E4 0} C_DIS
LIN {X -60.084, Y -146.4, Z 52.75, A 0, B 90, C 0, E1 0, E2 0, E3 0, E4 0} C_DIS
LIN {X -61.454, Y -138.499, Z 52.75, A 0, B 90, C 0, E1 0, E2 0, E3 0, E4 0} C_DIS
LIN {X -62.751, Y -130.585, Z 52.75, A 0, B 90, C 0, E1 0, E2 0, E3 0, E4 0} C_DIS
LIN {X -63.973, Y -122.66, Z 52.75, A 0, B 90, C 0, E1 0, E2 0, E3 0, E4 0} C_DIS
LIN {X -65.122, Y -114.724, Z 52.75, A 0, B 90, C 0, E1 0, E2 0, E3 0, E4 0} C_DIS
LIN {X -66.195, Y -106.777, Z 52.75, A 0, B 90, C 0, E1 0, E2 0, E3 0, E4 0} C_DIS
LIN {X -67.194, Y -98.82, Z 52.75, A 0, B 90, C 0, E1 0, E2 0, E3 0, E4 0} C_DIS
LIN {X -68.116, Y -90.855, Z 52.75, A 0, B 90, C 0, E1 0, E2 0, E3 0, E4 0} C_DIS
LIN {X -68.963, Y -82.881, Z 52.75, A 0, B 90, C 0, E1 0, E2 0, E3 0, E4 0} C_DIS
LIN {X -69.734, Y -74.899, Z 52.75, A 0, B 90, C 0, E1 0, E2 0, E3 0, E4 0} C_DIS
LIN {X -70.428, Y -66.91, Z 52.75, A 0, B 90, C 0, E1 0, E2 0, E3 0, E4 0} C_DIS
LIN {X -71.045, Y -58.915, Z 52.75, A 0, B 90, C 0, E1 0, E2 0, E3 0, E4 0} C_DIS
LIN {X -71.585, Y -50.914, Z 52.75, A 0, B 90, C 0, E1 0, E2 0, E3 0, E4 0} C_DIS
LIN {X -72.047, Y -42.908, Z 52.75, A 0, B 90, C 0, E1 0, E2 0, E3 0, E4 0} C_DIS
LIN {X -72.431, Y -34.899, Z 52.75, A 0, B 90, C 0, E1 0, E2 0, E3 0, E4 0} C_DIS
LIN {X -72.737, Y -26.886, Z 52.75, A 0, B 90, C 0, E1 0, E2 0, E3 0, E4 0} C_DIS
LIN {X -72.964, Y -18.87, Z 52.75, A 0, B 90, C 0, E1 0, E2 0, E3 0, E4 0} C_DIS
LIN {X -73.112, Y -10.852, Z 52.75, A 0, B 90, C 0, E1 0, E2 0, E3 0, E4 0} C_DIS
LIN {X -73.18, Y -2.834, Z 52.75, A 0, B 90, C 0, E1 0, E2 0, E3 0, E4 0} C_DIS
LIN {X -73.169, Y 5.185, Z 52.75, A 0, B 90, C 0, E1 0, E2 0, E3 0, E4 0} C_DIS
LIN {X -73.078, Y 13.204, Z 52.75, A 0, B 90, C 0, E1 0, E2 0, E3 0, E4 0} C_DIS
LIN {X -72.908, Y 21.221, Z 52.75, A 0, B 90, C 0, E1 0, E2 0, E3 0, E4 0} C_DIS
LIN {X -72.659, Y 29.236, Z 52.75, A 0, B 90, C 0, E1 0, E2 0, E3 0, E4 0} C_DIS
LIN {X -72.331, Y 37.248, Z 52.75, A 0, B 90, C 0, E1 0, E2 0, E3 0, E4 0} C_DIS
LIN {X -71.924, Y 45.257, Z 52.75, A 0, B 90, C 0, E1 0, E2 0, E3 0, E4 0} C_DIS
LIN {X -71.44, Y 53.261, Z 52.75, A 0, B 90, C 0, E1 0, E2 0, E3 0, E4 0} C_DIS
LIN {X -70.877, Y 61.26, Z 52.75, A 0, B 90, C 0, E1 0, E2 0, E3 0, E4 0} C_DIS
LIN {X -70.238, Y 69.254, Z 52.75, A 0, B 90, C 0, E1 0, E2 0, E3 0, E4 0} C_DIS
LIN {X -69.521, Y 77.241, Z 52.75, A 0, B 90, C 0, E1 0, E2 0, E3 0, E4 0} C_DIS
LIN {X -68.728, Y 85.22, Z 52.75, A 0, B 90, C 0, E1 0, E2 0, E3 0, E4 0} C_DIS
LIN {X -67.858, Y 93.192, Z 52.75, A 0, B 90, C 0, E1 0, E2 0, E3 0, E4 0} C_DIS
LIN {X -66.912, Y 101.155, Z 52.75, A 0, B 90, C 0, E1 0, E2 0, E3 0, E4 0} C_DIS
LIN {X -65.89, Y 109.108, Z 52.75, A 0, B 90, C 0, E1 0, E2 0, E3 0, E4 0} C_DIS
LIN {X -64.793, Y 117.052, Z 52.75, A 0, B 90, C 0, E1 0, E2 0, E3 0, E4 0} C_DIS
LIN {X -63.622, Y 124.985, Z 52.75, A 0, B 90, C 0, E1 0, E2 0, E3 0, E4 0} C_DIS
LIN {X -62.376, Y 132.906, Z 52.75, A 0, B 90, C 0, E1 0, E2 0, E3 0, E4 0} C_DIS
LIN {X -61.057, Y 140.816, Z 52.75, A 0, B 90, C 0, E1 0, E2 0, E3 0, E4 0} C_DIS
LIN {X -59.665, Y 148.713, Z 52.75, A 0, B 90, C 0, E1 0, E2 0, E3 0, E4 0} C_DIS
LIN {X -58.201, Y 156.597, Z 52.75, A 0, B 90, C 0, E1 0, E2 0, E3 0, E4 0} C_DIS
LIN {X -56.665, Y 164.468, Z 52.75, A 0, B 90, C 0, E1 0, E2 0, E3 0, E4 0} C_DIS
LIN {X -55.058, Y 172.324, Z 52.75, A 0, B 90, C 0, E1 0, E2 0, E3 0, E4 0} C_DIS
LIN {X -53.381, Y 180.166, Z 52.75, A 0, B 90, C 0, E1 0, E2 0, E3 0, E4 0} C_DIS
LIN {X -51.634, Y 187.992, Z 52.75, A 0, B 90, C 0, E1 0, E2 0, E3 0, E4 0} C_DIS
LIN {X -49.818, Y 195.803, Z 52.75, A 0, B 90, C 0, E1 0, E2 0, E3 0, E4 0} C_DIS
LIN {X -47.934, Y 203.597, Z 52.75, A 0, B 90, C 0, E1 0, E2 0, E3 0, E4 0} C_DIS
LIN {X -45.983, Y 211.375, Z 52.75, A 0, B 90, C 0, E1 0, E2 0, E3 0, E4 0} C_DIS
LIN {X -43.965, Y 219.136, Z 52.75, A 0, B 90, C 0, E1 0, E2 0, E3 0, E4 0} C_DIS
LIN {X -41.88, Y 226.879, Z 52.75, A 0, B 90, C 0, E1 0, E2 0, E3 0, E4 0} C_DIS
LIN {X -39.73, Y 234.605, Z 52.75, A 0, B 90, C 0, E1 0, E2 0, E3 0, E4 0} C_DIS
LIN {X -37.515, Y 242.312, Z 52.75, A 0, B 90, C 0, E1 0, E2 0, E3 0, E4 0} C_DIS
LIN {X -35.519, Y 250, Z 55.25, A 0, B 90, C 0, E1 0, E2 0, E3 0, E4 0} C_DIS
LIN {X -33.176, Y 257.648, Z 55.25, A 0, B 90, C 0, E1 0, E2 0, E3 0, E4 0} C_DIS
LIN {X -30.771, Y 265.277, Z 55.25, A 0, B 90, C 0, E1 0, E2 0, E3 0, E4 0} C_DIS
LIN {X -28.305, Y 272.886, Z 55.25, A 0, B 90, C 0, E1 0, E2 0, E3 0, E4 0} C_DIS
LIN {X -25.78, Y 280.476, Z 55.25, A 0, B 90, C 0, E1 0, E2 0, E3 0, E4 0} C_DIS
LIN {X -23.196, Y 288.046, Z 55.25, A 0, B 90, C 0, E1 0, E2 0, E3 0, E4 0} C_DIS
LIN {X -20.556, Y 295.597, Z 55.25, A 0, B 90, C 0, E1 0, E2 0, E3 0, E4 0} C_DIS
LIN {X -17.86, Y 303.128, Z 55.25, A 0, B 90, C 0, E1 0, E2 0, E3 0, E4 0} C_DIS
LIN {X -15.111, Y 310.64, Z 55.25, A 0, B 90, C 0, E1 0, E2 0, E3 0, E4 0} C_DIS
LIN {X -12.308, Y 318.132, Z 55.25, A 0, B 90, C 0, E1 0, E2 0, E3 0, E4 0} C_DIS
LIN {X -9.453, Y 325.604, Z 55.25, A 0, B 90, C 0, E1 0, E2 0, E3 0, E4 0} C_DIS
LIN {X -6.544, Y 333.055, Z 55.25, A 0, B 90, C 0, E1 0, E2 0, E3 0, E4 0} C_DIS
LIN {X -3.581, Y 340.485, Z 55.25, A 0, B 90, C 0, E1 0, E2 0, E3 0, E4 0} C_DIS
LIN {X -0.564, Y 347.893, Z 55.25, A 0, B 90, C 0, E1 0, E2 0, E3 0, E4 0} C_DIS
LIN {X 2.508, Y 355.279, Z 55.25, A 0, B 90, C 0, E1 0, E2 0, E3 0, E4 0} C_DIS
LIN {X 5.635, Y 362.641, Z 55.25, A 0, B 90, C 0, E1 0, E2 0, E3 0, E4 0} C_DIS
LIN {X 10.504, Y 368.708, Z 55.25, A 0, B 90, C 0, E1 0, E2 0, E3 0, E4 0} C_DIS
LIN {X 18.254, Y 368.659, Z 55.25, A 0, B 90, C 0, E1 0, E2 0, E3 0, E4 0} C_DIS
LIN {X 25.604, Y 365.504, Z 55.25, A 0, B 90, C 0, E1 0, E2 0, E3 0, E4 0} C_DIS
LIN {X 32.954, Y 362.349, Z 55.25, A 0, B 90, C 0, E1 0, E2 0, E3 0, E4 0} C_DIS
LIN {X 40.305, Y 359.194, Z 55.25, A 0, B 90, C 0, E1 0, E2 0, E3 0, E4 0} C_DIS
LIN {X 47.655, Y 356.039, Z 55.25, A 0, B 90, C 0, E1 0, E2 0, E3 0, E4 0} C_DIS
LIN {X 55.006, Y 352.884, Z 55.25, A 0, B 90, C 0, E1 0, E2 0, E3 0, E4 0} C_DIS
LIN {X 62.3, Y 349.615, Z 55.25, A 0, B 90, C 0, E1 0, E2 0, E3 0, E4 0} C_DIS
LIN {X 66.743, Y 343.35, Z 55.25, A 0, B 90, C 0, E1 0, E2 0, E3 0, E4 0} C_DIS
LIN {X 64.302, Y 335.821, Z 55.25, A 0, B 90, C 0, E1 0, E2 0, E3 0, E4 0} C_DIS
LIN {X 61.183, Y 328.456, Z 55.25, A 0, B 90, C 0, E1 0, E2 0, E3 0, E4 0} C_DIS
LIN {X 58.123, Y 321.065, Z 55.25, A 0, B 90, C 0, E1 0, E2 0, E3 0, E4 0} C_DIS
LIN {X 55.122, Y 313.651, Z 55.25, A 0, B 90, C 0, E1 0, E2 0, E3 0, E4 0} C_DIS
LIN {X 52.179, Y 306.213, Z 55.25, A 0, B 90, C 0, E1 0, E2 0, E3 0, E4 0} C_DIS
LIN {X 49.296, Y 298.751, Z 55.25, A 0, B 90, C 0, E1 0, E2 0, E3 0, E4 0} C_DIS
LIN {X 46.47, Y 291.268, Z 55.25, A 0, B 90, C 0, E1 0, E2 0, E3 0, E4 0} C_DIS
LIN {X 43.704, Y 283.763, Z 55.25, A 0, B 90, C 0, E1 0, E2 0, E3 0, E4 0} C_DIS
LIN {X 40.995, Y 276.236, Z 55.25, A 0, B 90, C 0, E1 0, E2 0, E3 0, E4 0} C_DIS
LIN {X 38.344, Y 268.689, Z 55.25, A 0, B 90, C 0, E1 0, E2 0, E3 0, E4 0} C_DIS
LIN {X 35.754, Y 261.121, Z 55.25, A 0, B 90, C 0, E1 0, E2 0, E3 0, E4 0} C_DIS
LIN {X 33.224, Y 253.533, Z 55.25, A 0, B 90, C 0, E1 0, E2 0, E3 0, E4 0} C_DIS
LIN {X 30.757, Y 245.924, Z 55.25, A 0, B 90, C 0, E1 0, E2 0, E3 0, E4 0} C_DIS
LIN {X 28.354, Y 238.294, Z 55.25, A 0, B 90, C 0, E1 0, E2 0, E3 0, E4 0} C_DIS
LIN {X 26.016, Y 230.645, Z 55.25, A 0, B 90, C 0, E1 0, E2 0, E3 0, E4 0} C_DIS
LIN {X 23.744, Y 222.975, Z 55.25, A 0, B 90, C 0, E1 0, E2 0, E3 0, E4 0} C_DIS
LIN {X 21.54, Y 215.286, Z 55.25, A 0, B 90, C 0, E1 0, E2 0, E3 0, E4 0} C_DIS
LIN {X 19.404, Y 207.577, Z 55.25, A 0, B 90, C 0, E1 0, E2 0, E3 0, E4 0} C_DIS
LIN {X 17.339, Y 199.849, Z 55.25, A 0, B 90, C 0, E1 0, E2 0, E3 0, E4 0} C_DIS
LIN {X 15.345, Y 192.103, Z 55.25, A 0, B 90, C 0, E1 0, E2 0, E3 0, E4 0} C_DIS
LIN {X 13.423, Y 184.338, Z 55.25, A 0, B 90, C 0, E1 0, E2 0, E3 0, E4 0} C_DIS
LIN {X 11.575, Y 176.556, Z 55.25, A 0, B 90, C 0, E1 0, E2 0, E3 0, E4 0} C_DIS
LIN {X 9.8, Y 168.756, Z 55.25, A 0, B 90, C 0, E1 0, E2 0, E3 0, E4 0} C_DIS
LIN {X 8.1, Y 160.94, Z 55.25, A 0, B 90, C 0, E1 0, E2 0, E3 0, E4 0} C_DIS
LIN {X 6.476, Y 153.108, Z 55.25, A 0, B 90, C 0, E1 0, E2 0, E3 0, E4 0} C_DIS
LIN {X 4.929, Y 145.26, Z 55.25, A 0, B 90, C 0, E1 0, E2 0, E3 0, E4 0} C_DIS
LIN {X 3.46, Y 137.397, Z 55.25, A 0, B 90, C 0, E1 0, E2 0, E3 0, E4 0} C_DIS
LIN {X 2.069, Y 129.52, Z 55.25, A 0, B 90, C 0, E1 0, E2 0, E3 0, E4 0} C_DIS
LIN {X 0.758, Y 121.629, Z 55.25, A 0, B 90, C 0, E1 0, E2 0, E3 0, E4 0} C_DIS
LIN {X -0.474, Y 113.725, Z 55.25, A 0, B 90, C 0, E1 0, E2 0, E3 0, E4 0} C_DIS
LIN {X -1.626, Y 105.81, Z 55.25, A 0, B 90, C 0, E1 0, E2 0, E3 0, E4 0} C_DIS
LIN {X -2.697, Y 97.883, Z 55.25, A 0, B 90, C 0, E1 0, E2 0, E3 0, E4 0} C_DIS
LIN {X -3.687, Y 89.945, Z 55.25, A 0, B 90, C 0, E1 0, E2 0, E3 0, E4 0} C_DIS
LIN {X -4.595, Y 81.998, Z 55.25, A 0, B 90, C 0, E1 0, E2 0, E3 0, E4 0} C_DIS
LIN {X -5.421, Y 74.042, Z 55.25, A 0, B 90, C 0, E1 0, E2 0, E3 0, E4 0} C_DIS
LIN {X -6.165, Y 66.077, Z 55.25, A 0, B 90, C 0, E1 0, E2 0, E3 0, E4 0} C_DIS
LIN {X -6.825, Y 58.106, Z 55.25, A 0, B 90, C 0, E1 0, E2 0, E3 0, E4 0} C_DIS
LIN {X -7.402, Y 50.128, Z 55.25, A 0, B 90, C 0, E1 0, E2 0, E3 0, E4 0} C_DIS
LIN {X -7.895, Y 42.144, Z 55.25, A 0, B 90, C 0, E1 0, E2 0, E3 0, E4 0} C_DIS
LIN {X -8.304, Y 34.155, Z 55.25, A 0, B 90, C 0, E1 0, E2 0, E3 0, E4 0} C_DIS
LIN {X -8.628, Y 26.163, Z 55.25, A 0, B 90, C 0, E1 0, E2 0, E3 0, E4 0} C_DIS
LIN {X -8.867, Y 18.168, Z 55.25, A 0, B 90, C 0, E1 0, E2 0, E3 0, E4 0} C_DIS
LIN {X -9.021, Y 10.17, Z 55.25, A 0, B 90, C 0, E1 0, E2 0, E3 0, E4 0} C_DIS
LIN {X -9.089, Y 2.171, Z 55.25, A 0, B 90, C 0, E1 0, E2 0, E3 0, E4 0} C_DIS
LIN {X -9.071, Y -5.827, Z 55.25, A 0, B 90, C 0, E1 0, E2 0, E3 0, E4 0} C_DIS
LIN {X -8.967, Y -13.826, Z 55.25, A 0, B 90, C 0, E1 0, E2 0, E3 0, E4 0} C_DIS
LIN {X -8.777, Y -21.822, Z 55.25, A 0, B 90, C 0, E1 0, E2 0, E3 0, E4 0} C_DIS
LIN {X -8.502, Y -29.817, Z 55.25, A 0, B 90, C 0, E1 0, E2 0, E3 0, E4 0} C_DIS
LIN {X -8.141, Y -37.808, Z 55.25, A 0, B 90, C 0, E1 0, E2 0, E3 0, E4 0} C_DIS
LIN {X -7.696, Y -45.794, Z 55.25, A 0, B 90, C 0, E1 0, E2 0, E3 0, E4 0} C_DIS
